	IF ncounter = nCount THEN 
		FOR i := 0 TO SIZEOF(refArray)-1 BY 1 DO 
			refArray[i] := FALSE;
		END_FOR
		F_checkMoveFinish := TRUE;
	ELSE
		F_checkMoveFinish := FALSE;
	END_IF
ELSE
	FOR i := 0 TO SIZEOF(refArray)-1 BY 1 DO 
			refArray[i] := FALSE;
		END_FOR
		F_checkMoveFinish := TRUE;
END_IF

END_FUNCTION

// ---- POUs/PROGRAMS/eflex.TcPOU
PROGRAM eflex
VAR
fbMqttClient	: FB_IotMqttClient;


bSetParameter 	: BOOL := TRUE;
bConnect 		: BOOL := TRUE;

(* published message *)
bPublish 		: BOOL;
sTopicPub 		: STRING(255) := 'flipper2.1toNodeRed'; //Publish topic. Must match syntax of nodeRed "mqtt out - topic"
sPayloadPub 	: STRING (255):= 'This is a test';
x				: UDINT;

(* recieved message *)
bSubscribed 	: BOOL;
sTopicSub 		: STRING(255) := 'toFlipper2.1PLC'; //Suscribe topic. Must match syntax of nodeRed "mqtt in - topic"
sTopicRcv 		: STRING(255);
sPayloadRcv 	: STRING(255);

fbMessageQueue	: FB_IotMqttMessageQueue;
fbMessage		: FB_IotMqttMessage;
fbJsonDataType 	: FB_JsonReadWriteDataType;
eflexMsgIn 		: ST_eflexMsgIn; //Custom Data Structure that must match variable types of eflex variables being sent through nodeRed. 
sBuffer 		: STRING(255);
END_VAR

IF bSetParameter THEN
	bSetParameter 				:= FALSE;
	fbMqttClient.sHostName 		:= '10.0.0.41';
	fbMqttClient.nHostPort 		:= 1883;
	fbMqttClient.sUserName 		:= 'eflex';
	fbMqttClient.sUserPassword 	:= 'dean-wormwood-sway-lope';
	fbMqttClient.ipMessageQueue := fbMessageQueue;
END_IF

fbMqttClient.Execute(bConnect);


IF fbMqttClient.bConnected THEN
	IF NOT bSubscribed THEN
		bSubscribed 	:= fbMqttClient.Subscribe(sTopic := sTopicSub, eQoS:= TcIOTMqttQos.AtMostOnceDelivery);
	END_IF
	IF bPublish THEN
		fbMqttClient.Publish(
		sTopic			:= sTopicPub, 
		pPayload		:= ADR(sBuffer), 
		nPayloadSize	:= LEN2(ADR(sBuffer)), 
		eQoS			:= TcIOTMqttQos.AtMostOnceDelivery, 
		bRetain			:= FALSE, 
		bQueue			:= FALSE);
		bPublish 		:= FALSE;	
		x := MEMSET(destAddr := ADR(sPayloadRcv),fillByte := 0,n := SIZEOF(sPayloadRcv));			
	END_IF
END_IF

IF fbMessageQueue.nQueuedMessages > 0 THEN 
	IF fbMessageQueue.Dequeue(fbMessage := fbMessage) THEN
		fbMessage.GetTopic(pTopic := ADR(sTopicRcv), nTopicSize := SIZEOF(sTopicRcv));
		fbMessage.GetPayload(pPayload:=ADR(sPayloadRcv), nPayloadSize:=SIZEOF(sPayloadRcv), bSetNullTermination:=FALSE);
		fbJsonDataType.SetSymbolFromJson(sPayloadRcv,'ST_eflexMsgIn',SIZEOF(eflexMsgIn), ADR(eflexMsgIn));
		GVL_eflex.bEflexPresent := TRUE;
		GVL_eflex.fFlipHeight := eflexMsgIn.flipHeight;
		GVL_eflex.fStudHeight := eflexMsgIn.studHeight;
		GVL_eflex.sSpaModel := eflexMsgIn.spaModel;
		GVL_eflex.fBaseInHeight := eflexMsgIn.baseInHeight;
		GVL_eflex.fSpaOutHeight := eflexMsgIn.spaOutHeight;
		sBuffer := fbJsonDataType.GetJsonStringFromSymbol('ST_eflexMsgIn',SIZEOF(eflexMsgIn), ADR(eflexMsgIn));
		bPublish := TRUE;
	END_IF
END_IF

IF GVL_eflex.bEflexPresent THEN
	IF GVL_eflex.fFlipHeight < 1 OR GVL_eflex.fStudHeight < 1 OR GVL_eflex.sSpaModel = '' THEN
		GVL_eflex.sSpaModel := 'ERROR';
	END_IF
END_IF

END_PROGRAM

// ---- POUs/PROGRAMS/tempEflex.TcPOU
PROGRAM tempEflex
VAR
	//HMI
	nEflexState : INT;
END_VAR



CASE nEflexState OF 
	0://Steady State
	1://A5L
		GVL_eflex.fBaseInHeight := 30;
		GVL_eflex.fSpaOutHeight := 35;
		GVL_eflex.fFlipHeight := 19;
		GVL_eflex.fStudHeight := 7;
		GVL_eflex.sSpaModel := 'A5L';
		GVL_eflex.bEflexPresent := TRUE;
		nEflexState := 0;
	2://A6
		GVL_eflex.fBaseInHeight := 30;
		GVL_eflex.fSpaOutHeight := 35;
		GVL_eflex.fFlipHeight := 22;
		GVL_eflex.fStudHeight := 12;
		GVL_eflex.sSpaModel := 'A6';
		GVL_eflex.bEflexPresent := TRUE;
		nEflexState := 0;
	3://A7
		GVL_eflex.fBaseInHeight := 30;
		GVL_eflex.fSpaOutHeight := 35;
		GVL_eflex.fFlipHeight := 23;
		GVL_eflex.fStudHeight := 12;
		GVL_eflex.sSpaModel := 'A7';
		GVL_eflex.bEflexPresent := TRUE;
		nEflexState := 0;
	4://A8
		GVL_eflex.fBaseInHeight := 27.5;
		GVL_eflex.fSpaOutHeight := 35;
		GVL_eflex.fFlipHeight := 24;
		GVL_eflex.fStudHeight := 15.5;
		GVL_eflex.sSpaModel := 'A8';
		GVL_eflex.bEflexPresent := TRUE;
		nEflexState := 0;
	5://A9L
		GVL_eflex.fBaseInHeight := 20.5;
		GVL_eflex.fSpaOutHeight := 35;
		GVL_eflex.fFlipHeight := 24;
		GVL_eflex.fStudHeight := 14.5;
		GVL_eflex.sSpaModel := 'A9L';
		GVL_eflex.bEflexPresent := TRUE;
		nEflexState := 0;
END_CASE

END_PROGRAM

// ---- POUs/PROGRAMS/motorsInit.TcPOU
PROGRAM motorsInit
VAR
	nInitCount	: INT;
	bChecked 	: BOOL := FALSE;
	nWaitCount 	: INT;
	aMoveFinish	: ARRAY[0..10] OF BOOL; // Can track the completion of up to 10 simultaneous moves
	fbMotorTimeOut : TON;
	fbWaitInit : TON;
	bMotorsInit : BOOL;
END_VAR

	updateMotors();
bMotorsInit := FALSE;
fbWaitInit(IN:= TRUE, PT:=T#3S);
fbMotorTimeOut(PT:=T#1M);

IF fbWaitInit.Q THEN
		GVL_machine.bMotorInitFailedDisp := FALSE;
		
		IF NOT aMoveFinish[1] THEN
			aMoveFinish[1] := GVL_devices.fbColumn1Motor.init(
								bMotorInvertedIn:= TRUE, 
								bMotorDisablesIn:= FALSE, 
								fMoveAcclIn:= 200, 
								fMoveDclIn:= 200, 
								fMoveVelocityIn:= 10, 
								torqueVelocityIn:= 10, 
								torqueAccelerationIn:= 50, 
								torqueDecelerationIn:= 50, 
								homeVelocityIn:= 7, 
								homeSetPositionIn:= 0, 
								homeTorqueLimitIn:= 8,
								jogTorqueIn := 100,
								bHasHomeSensorIn := FALSE);
		END_IF
		IF NOT aMoveFinish[2] THEN
			aMoveFinish[2] := GVL_devices.fbColumn2Motor.init(
								bMotorInvertedIn:= TRUE, 
								bMotorDisablesIn:= FALSE, 
								fMoveAcclIn:= 200, 
								fMoveDclIn:= 200, 
								fMoveVelocityIn:= 10, 
								torqueVelocityIn:= 10, 
								torqueAccelerationIn:= 50, 
								torqueDecelerationIn:= 50, 
								homeVelocityIn:= 7, 
								homeSetPositionIn:= 0, 
								homeTorqueLimitIn:= 8,
								jogTorqueIn := 100,
								bHasHomeSensorIn := TRUE);
		END_IF
		IF NOT aMoveFinish[3] THEN
			aMoveFinish[3] := GVL_devices.fbColumn3Motor.init(
								bMotorInvertedIn:= TRUE, 
								bMotorDisablesIn:= FALSE, 
								fMoveAcclIn:= 200, 
								fMoveDclIn:= 200, 
								fMoveVelocityIn:= 10, 
								torqueVelocityIn:= 10, 
								torqueAccelerationIn:= 50, 
								torqueDecelerationIn:= 50, 
								homeVelocityIn:= 7, 
								homeSetPositionIn:= 0, 
								homeTorqueLimitIn:= 8,
								jogTorqueIn := 100,
								bHasHomeSensorIn := FALSE);
		END_IF
		IF NOT aMoveFinish[4] THEN
			aMoveFinish[4] := GVL_devices.fbLftClampMotor.init(
								bMotorInvertedIn:= TRUE, 
								bMotorDisablesIn:= TRUE, 
								fMoveAcclIn:= 100, 
								fMoveDclIn:= 100, 
								fMoveVelocityIn:= 20, 
								torqueVelocityIn:= 7, 
								torqueAccelerationIn:= 100, 
								torqueDecelerationIn:= 100, 
								homeVelocityIn:= 10, 
								homeSetPositionIn:= 0, 
								homeTorqueLimitIn:= 20,
								jogTorqueIn := GVL_persistent.fTempLftClampTorque,
								bHasHomeSensorIn := FALSE);
		END_IF
		IF NOT aMoveFinish[5] THEN
			aMoveFinish[5] := GVL_devices.fbRhtClampMotor.init(
								bMotorInvertedIn:= FALSE, 
								bMotorDisablesIn:= TRUE, 
								fMoveAcclIn:= 100, 
								fMoveDclIn:= 100, 
								fMoveVelocityIn:= 20, 
								torqueVelocityIn:= 7, 
								torqueAccelerationIn:= 100, 
								torqueDecelerationIn:= 100, 
								homeVelocityIn:= 10, 
								homeSetPositionIn:= 0, 
								homeTorqueLimitIn:= 40,
								jogTorqueIn := GVL_persistent.fClampOnTorque,
								bHasHomeSensorIn := FALSE);
		END_IF
		IF NOT aMoveFinish[6] THEN
			aMoveFinish[6] := GVL_devices.fbLftRotationMotor.init(
								bMotorInvertedIn:= TRUE, 
								bMotorDisablesIn:= TRUE, 
								fMoveAcclIn:= 50, 
								fMoveDclIn:= 50, 
								fMoveVelocityIn:= 8, 
								torqueVelocityIn:= 7, 
								torqueAccelerationIn:= 50, 
								torqueDecelerationIn:= 50, 
								homeVelocityIn:= 3, 
								homeSetPositionIn:= GVL_persistent.fLftRotationHomePos, 
								homeTorqueLimitIn:= 20,
								jogTorqueIn := 100,
								bHasHomeSensorIn := FALSE);
		END_IF
		IF NOT aMoveFinish[7] THEN
			aMoveFinish[7] := GVL_devices.fbRhtRotationMotor.init(
								bMotorInvertedIn:= FALSE, 
								bMotorDisablesIn:= TRUE, 
								fMoveAcclIn:= 50, 
								fMoveDclIn:= 50, 
								fMoveVelocityIn:= 8, 
								torqueVelocityIn:= 7, 
								torqueAccelerationIn:= 50, 
								torqueDecelerationIn:= 50, 
								homeVelocityIn:= 3, 
								homeSetPositionIn:= GVL_persistent.fRhtRotationHomePos,
								homeTorqueLimitIn:= 20,
								jogTorqueIn := 100,
								bHasHomeSensorIn := FALSE);
		END_IF
		IF NOT aMoveFinish[8] THEN
			aMoveFinish[8] := GVL_devices.fbLftWidthMotor.init(
								bMotorInvertedIn:= FALSE, 
								bMotorDisablesIn:= TRUE, 
								fMoveAcclIn:= 50, 
								fMoveDclIn:= 50, 
								fMoveVelocityIn:= 20, 
								torqueVelocityIn:= 20, 
								torqueAccelerationIn:= 50, 
								torqueDecelerationIn:= 50, 
								homeVelocityIn:= 10, 
								homeSetPositionIn:= 0, 
								homeTorqueLimitIn:= 15,
								jogTorqueIn := 30,
								bHasHomeSensorIn := TRUE);
		END_IF
		IF NOT aMoveFinish[9] THEN
			aMoveFinish[9] := GVL_devices.fbRhtWidthMotor.init(
								bMotorInvertedIn:= FALSE, 
								bMotorDisablesIn:= TRUE, 
								fMoveAcclIn:= 50, 
								fMoveDclIn:= 50, 
								fMoveVelocityIn:= 20, 
								torqueVelocityIn:= 20, 
								torqueAccelerationIn:= 50, 
								torqueDecelerationIn:= 50, 
								homeVelocityIn:= 10, 
								homeSetPositionIn:= 0, 
								homeTorqueLimitIn:= 15,
								jogTorqueIn := 30,
								bHasHomeSensorIn := TRUE);
		END_IF
		IF NOT aMoveFinish[0] THEN
			aMoveFinish[0] := GVL_devices.fbColumn0Motor.init(
								bMotorInvertedIn:= TRUE, 
								bMotorDisablesIn:= FALSE, 
								fMoveAcclIn:= 200, 
								fMoveDclIn:= 200, 
								fMoveVelocityIn:= 10, 
								torqueVelocityIn:= 10, 
								torqueAccelerationIn:= 50, 
								torqueDecelerationIn:= 50, 
								homeVelocityIn:= 7, 
								homeSetPositionIn:= 0, 
								homeTorqueLimitIn:= 8,
								jogTorqueIn := 100,
								bHasHomeSensorIn := TRUE);
		END_IF
		
		IF F_checkMoveFinish(aMoveFinish,10,FALSE) THEN
			GVL_machine.sMotorInitState := 'PASSED';
			fbWaitInit(IN := FALSE);
			fbMotorTimeOut(IN := FALSE);
			GVL_machine.bMotorInitFailedDisp := FALSE;
			GVL_machine.bMotorsInitialized := TRUE;
			bMotorsInit := TRUE;
		ELSE // Start Timeout Timer
			fbMotorTimeout.IN := TRUE;
			IF fbMotorTimeout.Q THEN
				fbWaitInit(IN := FALSE);
				fbMotorTimeOut(IN := FALSE);
				GVL_machine.sMotorInitState := 'FAILED';
				GVL_machine.bMotorInitFailedDisp := TRUE;
				F_checkMoveFinish(aMoveFinish,10,TRUE);
				GVL_machine.bMotorsInitialized := TRUE;
			END_IF
		END_IF
	IF LEN(GVL_machine.sMotorInitState) <> 0 THEN
		GVL_devices.fbLftClampMotor.brakeOn();
		GVL_devices.fbRhtClampMotor.brakeOn();
	END_IF
END_IF

END_PROGRAM

// ---- POUs/PROGRAMS/updateMotors.TcPOU
PROGRAM updateMotors
VAR
END_VAR

GVL_devices.fbLftWidthMotor();
GVL_devices.fbRhtWidthMotor();

GVL_devices.fbLftClampMotor();
GVL_devices.fbRhtClampMotor();

GVL_devices.fbLftRotationMotor();	
GVL_devices.fbRhtRotationMotor();	

GVL_devices.fbColumn0Motor();	
GVL_devices.fbColumn1Motor();	
GVL_devices.fbColumn2Motor();	
GVL_devices.fbColumn3Motor();

END_PROGRAM

// ---- POUs/PROGRAMS/manual.TcPOU
PROGRAM manual
VAR
	aMoveFinishRotation			: ARRAY[0..10] OF BOOL; // Can track the completion of up to 10 simultaneous moves
	aMoveFinishColumn			: ARRAY[0..10] OF BOOL; // Can track the completion of up to 10 simultaneous moves
	aMoveFinishClamping			: ARRAY[0..10] OF BOOL; // Can track the completion of up to 10 simultaneous moves
	aMoveFinishWidth			: ARRAY[0..10] OF BOOL; // Can track the completion of up to 10 simultaneous moves
	
	eRotationState 	: E_manualState;
	eColumnState 	: E_manualState;
	eClampingState	: E_manualState;
	eWidthState		: E_manualState;
	eTableState		: E_manualState;
	
	fbCoupledRotation : TON;
	fbCoupledColumn : TON;
	fbCoupledClamping : TON;
	fbCoupledWidth : TON;
	tUncoupledTimeout : TIME := T#500MS;
	
	bRotationStopped 	: BOOL;
	bColumnStopped 		: BOOL;
	bClampingStopped 	: BOOL;
	bWidthStopped 		: BOOL;
	bTableStopped		: BOOL;
	
	//HMI 
	bHideRotationBtns 	: BOOL;
	bHideColumnBtns 	: BOOL;
	bHideClampingBtns	: BOOL;
	bHideWidthBtns		: BOOL;
	bHideTableBtns		: BOOL;
	
	bRotationMoveStatus : BOOL; // True- error is present
	bColumnMoveStatus 	: BOOL;
	bClampingMoveStatus : BOOL;
	bWidthMoveStatus 	: BOOL;
	bTableMoveStatus 	: BOOL;
	writeParameter		: MC_AxisParameter;
END_VAR

// Both manualScreen and manualBypassedScreen use this program for their functionality. Only difference is buttons are not hidden on manualBypassedScreen. 
///////////////////////// PAGE CHANGE TO MANUAL //////////////////////////////
IF GVL_machine.bPageChange THEN 
	eRotationState 	:= STEADYSTATE;
	eColumnState 	:= STEADYSTATE;
	eClampingState 	:= STEADYSTATE;
	eWidthState 	:= STEADYSTATE;
	eTableState		:= STEADYSTATE;
	GVL_machine.bPageChange	:= FALSE;
END_IF

fbCoupledRotation(PT := tUncoupledTimeout);
fbCoupledColumn(PT := tUncoupledTimeout); 
fbCoupledClamping (PT := tUncoupledTimeout);
fbCoupledWidth (PT := tUncoupledTimeout);


IF GVL_machine.bMuteSafety OR GVL_machine.bSafetyBypass THEN
	//pass -default is yellow
ELSIF bRotationStopped AND bColumnStopped AND bClampingStopped AND bWidthStopped AND bTableStopped THEN
	GVL_devices.fbLtCurtains.mute();
	IF GVL_devices.fbLtCurtains.curtainsMuted THEN
		GVL_devices.fbLtBars.greenOn();
	END_IF
ELSIF NOT bRotationStopped OR NOT bColumnStopped OR NOT bClampingStopped OR NOT bWidthStopped OR NOT bTableStopped THEN
	GVL_devices.fbLtBars.redOn();
END_IF




IF NOT GVL_machine.bSafetyOk AND NOT GVL_machine.bSafetyBypass THEN 
	GVL_devices.fbLtBars.redOn();
	GVL_devices.fbColumn0Motor.estop();
	GVL_devices.fbColumn1Motor.estop();
	GVL_devices.fbColumn2Motor.estop();
	GVL_devices.fbColumn3Motor.estop();
	GVL_devices.fbLftClampMotor.estop();
	GVL_devices.fbRhtClampMotor.estop();
	GVL_devices.fbLftRotationMotor.estop();
	GVL_devices.fbRhtRotationMotor.estop();
	GVL_devices.fbLftWidthMotor.estop();
	GVL_devices.fbRhtWidthMotor.estop();
	GVL_devices.fbTable.estop();
	eRotationState 	:= STEADYSTATE;
	eColumnState 	:= STEADYSTATE;
	eClampingState 	:= STEADYSTATE;
	eWidthState 	:= STEADYSTATE;
	
ELSE // No Estop or Light Curtain 
	(*				Rotation Motion 			*)
		bRotationStopped := FALSE;
		bHideRotationBtns := TRUE;
		CASE eRotationState OF 
			STEADYSTATE:
				bHideRotationBtns := FALSE;
				bRotationStopped := TRUE;
				fbCoupledRotation.IN := FALSE;
				bRotationMoveStatus := FALSE;
				F_checkMoveFinish(aMoveFinishRotation,1,TRUE);
				
			MOVEAWAYDIRECTION:
				bHideRotationBtns := FALSE;
				CASE GVL_devices.fbLftRotationMotor.moveToJog(0) OF 
					1: // Good
					13://Error
						bRotationMoveStatus := TRUE; 
						GVL_machine.motorErrorList := LFTROTATION;
						GVL_machine.bErrorPresent := TRUE;
				END_CASE
				CASE GVL_devices.fbRhtRotationMotor.moveToJog(1) OF
					1: // Good
					13://Error
						bRotationMoveStatus := TRUE;
						GVL_machine.motorErrorList := RHTROTATION;
						GVL_machine.bErrorPresent := TRUE; 
				END_CASE
				CASE F_checkCoupledMovement(GVL_devices.fbLftRotationMotor.fbMotor,GVL_devices.fbRhtRotationMotor.fbMotor) OF 
						0: fbCoupledRotation.IN := FALSE;
						1,2: fbCoupledRotation.IN := TRUE;
						3: fbCoupledRotation.IN := FALSE;
				END_CASE
				
			MOVEHOMEDIRECTION:
				bHideRotationBtns := FALSE;
				CASE GVL_devices.fbLftRotationMotor.moveToJog(1) OF
					1: // Good
					13://Error
						bRotationMoveStatus := TRUE;
						GVL_machine.motorErrorList := LFTROTATION;
						GVL_machine.bErrorPresent := TRUE; 
				END_CASE
				CASE GVL_devices.fbRhtRotationMotor.moveToJog(0) OF
					1: // Good
					13://Error
						bRotationMoveStatus := TRUE; 
						GVL_machine.motorErrorList := RHTROTATION;
						GVL_machine.bErrorPresent := TRUE; 
				END_CASE
				CASE F_checkCoupledMovement(GVL_devices.fbLftRotationMotor.fbMotor,GVL_devices.fbRhtRotationMotor.fbMotor) OF 
						0: fbCoupledRotation.IN := FALSE;
						1,2: fbCoupledRotation.IN := TRUE;
						3: fbCoupledRotation.IN := FALSE;
				END_CASE
				
			RESET:
				IF NOT aMoveFinishRotation[0] THEN
					CASE GVL_devices.fbLftRotationMotor.reset() OF
						1:// Done
							aMoveFinishRotation[0] := TRUE;
						13:// Error
							bRotationMoveStatus := TRUE;
							GVL_machine.motorErrorList := LFTROTATION;
							GVL_machine.bErrorPresent := TRUE;
					END_CASE
				END_IF
				IF NOT aMoveFinishRotation[1] THEN
					CASE GVL_devices.fbRhtRotationMotor.reset() OF
						1:// Done
							aMoveFinishRotation[1] := TRUE;
						13:// Error
							bRotationMoveStatus := TRUE;
							GVL_machine.motorErrorList := RHTROTATION;
							GVL_machine.bErrorPresent := TRUE; 
						
					END_CASE 
				END_IF
				IF F_checkMoveFinish(aMoveFinishRotation,2,FALSE) THEN
					bRotationMoveStatus := FALSE;
					eRotationState := STEADYSTATE;
				END_IF
				
			HOMING:
				IF GVL_devices.fbLftRotationMotor.fbMotor.Status.Homed AND GVL_devices.fbRhtRotationMotor.fbMotor.Status.Homed THEN
					CASE F_checkCoupledMovement(GVL_devices.fbLftRotationMotor.fbMotor,GVL_devices.fbRhtRotationMotor.fbMotor) OF 
						0: fbCoupledRotation.IN := FALSE;
						1,2: fbCoupledRotation.IN := TRUE;
						3: fbCoupledRotation.IN := FALSE;
					END_CASE
				END_IF
				IF NOT aMoveFinishRotation[0] THEN
					CASE GVL_devices.fbLftRotationMotor.homeToTorque() OF 
						1:// Done
							aMoveFinishRotation[0] := TRUE;
						13:// Error
							GVL_machine.motorErrorList := LFTROTATION;
							GVL_machine.bErrorPresent := TRUE;
					END_CASE
				END_IF
				IF NOT aMoveFinishRotation[1] THEN
					CASE GVL_devices.fbRhtRotationMotor.homeToTorque() OF 
						1:// Done
							aMoveFinishRotation[1] := TRUE;
						13:// Error
							GVL_machine.motorErrorList := RHTROTATION;
							GVL_machine.bErrorPresent := TRUE; 
					END_CASE
				END_IF
				IF F_checkMoveFinish(aMoveFinishRotation,2,FALSE) THEN
					eRotationState := STEADYSTATE;
				END_IF
		END_CASE
		
		//Initial Homing not done or Components not moving together
		IF NOT GVL_devices.fbLftRotationMotor.fbMotor.Status.Homed OR NOT GVL_devices.fbRhtRotationMotor.fbMotor.Status.Homed OR fbCoupledRotation.Q OR bRotationMoveStatus THEN	
			GVL_devices.fbLftRotationMotor.estop();
			GVL_devices.fbRhtRotationMotor.estop();
			bHideRotationBtns := TRUE;
		END_IF
		
	(*				Column Motion 				*)
		bColumnStopped := FALSE;
		bHideColumnBtns := TRUE;
		CASE eColumnState OF 
			STEADYSTATE:
				bHideColumnBtns := FALSE;
				bColumnStopped := TRUE;
				fbCoupledColumn.IN := FALSE;
				bColumnMoveStatus := FALSE;
				F_checkMoveFinish(aMoveFinishColumn,1,TRUE);
				
			MOVEAWAYDIRECTION:
				bHideColumnBtns := FALSE;
				IF GVL_devices.fbColumn1Motor.fbMotor.Status.Coupled AND GVL_devices.fbColumn2Motor.fbMotor.Status.Coupled AND GVL_devices.fbColumn3Motor.fbMotor.Status.Coupled THEN
					GVL_devices.fbColumn0Motor.motorIdle := FALSE;
					GVL_devices.fbColumn1Motor.motorIdle := FALSE;
					GVL_devices.fbColumn2Motor.motorIdle := FALSE;
					GVL_devices.fbColumn3Motor.motorIdle := FALSE;
					CASE GVL_devices.fbColumn0Motor.moveToJog(0) OF
						1:// Good
						13:// Error
							bColumnMoveStatus := TRUE;
							GVL_machine.motorErrorList := COLUMN0;
							GVL_machine.bErrorPresent := TRUE; 
					END_CASE
				ELSE // Couple Motors
					GVL_devices.fbColumn1Motor.coupleToAxis(GVL_devices.fbColumn0Motor.fbMotor);
					GVL_devices.fbColumn2Motor.coupleToAxis(GVL_devices.fbColumn0Motor.fbMotor);
					GVL_devices.fbColumn3Motor.coupleToAxis(GVL_devices.fbColumn0Motor.fbMotor);
				END_IF
				
			MOVEHOMEDIRECTION:
				bHideColumnBtns := FALSE;
				
				
				IF GVL_devices.fbColumn1Motor.fbMotor.Status.Coupled AND GVL_devices.fbColumn2Motor.fbMotor.Status.Coupled AND GVL_devices.fbColumn3Motor.fbMotor.Status.Coupled THEN
					GVL_devices.fbColumn0Motor.motorIdle := FALSE;
					GVL_devices.fbColumn1Motor.motorIdle := FALSE;
					GVL_devices.fbColumn2Motor.motorIdle := FALSE;
					GVL_devices.fbColumn3Motor.motorIdle := FALSE;
					CASE GVL_devices.fbColumn0Motor.moveToJog(1) OF 
						1:// Good
						13:// Error
							bColumnMoveStatus := TRUE;
							GVL_machine.motorErrorList := COLUMN0;
							GVL_machine.bErrorPresent := TRUE; 
					END_CASE
				ELSE // Couple Motors
					GVL_devices.fbColumn1Motor.coupleToAxis(GVL_devices.fbColumn0Motor.fbMotor);
					GVL_devices.fbColumn2Motor.coupleToAxis(GVL_devices.fbColumn0Motor.fbMotor);
					GVL_devices.fbColumn3Motor.coupleToAxis(GVL_devices.fbColumn0Motor.fbMotor);
				END_IF
			RESET:
				IF NOT aMoveFinishColumn[0] THEN
					CASE GVL_devices.fbColumn0Motor.reset() OF 
						1:// Done
							aMoveFinishColumn[0] := TRUE;
						13:// Error
							bColumnMoveStatus := TRUE;
							GVL_machine.motorErrorList := COLUMN0;
							GVL_machine.bErrorPresent := TRUE; 
					END_CASE
				END_IF
				IF NOT aMoveFinishColumn[1] THEN
					CASE GVL_devices.fbColumn1Motor.reset() OF 
						1:// Done
							aMoveFinishColumn[1] := TRUE;
						13:// Error
							bColumnMoveStatus := TRUE;
							GVL_machine.motorErrorList := COLUMN1;
							GVL_machine.bErrorPresent := TRUE; 
					END_CASE
				END_IF
				IF NOT aMoveFinishColumn[2] THEN
					CASE GVL_devices.fbColumn2Motor.reset() OF 
						1:// Done
							aMoveFinishColumn[2] := TRUE;
						13:// Error
							bColumnMoveStatus := TRUE;
							GVL_machine.motorErrorList := COLUMN2;
							GVL_machine.bErrorPresent := TRUE; 
					END_CASE
				END_IF
				IF NOT aMoveFinishColumn[3] THEN
					CASE GVL_devices.fbColumn3Motor.reset() OF 
						1:// Done
							aMoveFinishColumn[3] := TRUE;
						13:// Error
							bColumnMoveStatus := TRUE;
							GVL_machine.motorErrorList := COLUMN3;
							GVL_machine.bErrorPresent := TRUE; 
					END_CASE
				END_IF
				
				IF F_checkMoveFinish(aMoveFinishColumn,4,FALSE) THEN
					eColumnState := STEADYSTATE;
				END_IF
				
			HOMING:
				(*IF GVL_devices.fbColumn0Motor.fbMotor.Status.Homed AND GVL_devices.fbColumn2Motor.fbMotor.Status.Homed THEN
					writeParameter := AxisMaxSoftPosLimit;
					IF NOT aMoveFinishColumn[0] THEN
						CASE GVL_devices.fbColumn2Motor.writeRealParameter(writeParameter,1) OF 
							1: //Done
								aMoveFinishColumn[0] := TRUE;
							13:// Error
								bColumnMoveStatus := TRUE;
								GVL_machine.motorErrorList := COLUMN2;
								GVL_machine.bErrorPresent := TRUE; 
						END_CASE
					END_IF
					IF aMoveFinishColumn[0] AND NOT aMoveFinishColumn[1] THEN
						IF GVL_devices.fbColumn1Motor.fbMotor.Status.Coupled AND GVL_devices.fbColumn2Motor.fbMotor.Status.Coupled AND GVL_devices.fbColumn3Motor.fbMotor.Status.Coupled THEN
							GVL_devices.fbColumn0Motor.motorIdle := FALSE;
							GVL_devices.fbColumn1Motor.motorIdle := FALSE;
							GVL_devices.fbColumn2Motor.motorIdle := FALSE;
							GVL_devices.fbColumn3Motor.motorIdle := FALSE;
							CASE GVL_devices.fbColumn0Motor.homeToSensor(0) OF 
								1: // Done
									aMoveFinishColumn[1] := TRUE;
								13:// Error
									bColumnMoveStatus := TRUE;
									GVL_machine.motorErrorList := COLUMN0;
									GVL_machine.bErrorPresent := TRUE; 
							END_CASE
						ELSE // Couple Motors to Column0
							GVL_devices.fbColumn1Motor.coupleToAxis(GVL_devices.fbColumn0Motor.fbMotor);
							GVL_devices.fbColumn2Motor.coupleToAxis(GVL_devices.fbColumn0Motor.fbMotor);
							GVL_devices.fbColumn3Motor.coupleToAxis(GVL_devices.fbColumn0Motor.fbMotor);
						END_IF
					END_IF
					IF aMoveFinishColumn[1] AND NOT aMoveFinishColumn[2] THEN
						CASE GVL_devices.fbColumn2Motor.writeRealParameter(writeParameter,0) OF 
							1:// Done
								aMoveFinishColumn[2] := TRUE;
							13://Error
								bColumnMoveStatus := TRUE;
								GVL_machine.motorErrorList := COLUMN2;
								GVL_machine.bErrorPresent := TRUE; 
						END_CASE
					END_IF
					IF F_checkMoveFinish(aMoveFinishColumn,3,FALSE) THEN
						eColumnState := STEADYSTATE;
					END_IF
				ELSE
					IF NOT aMoveFinishColumn[0] THEN
						IF GVL_devices.fbColumn1Motor.fbMotor.Status.Coupled THEN
							GVL_devices.fbColumn0Motor.motorIdle := FALSE;
							GVL_devices.fbColumn1Motor.motorIdle := FALSE;
							CASE GVL_devices.fbColumn0Motor.homeToSensor(0) OF 
								1:// Done
									aMoveFinishColumn[0] := TRUE;
								13:// Error
									bColumnMoveStatus := TRUE;
									GVL_machine.motorErrorList := COLUMN0;
									GVL_machine.bErrorPresent := TRUE; 
							END_CASE
						ELSE
							GVL_devices.fbColumn1Motor.coupleToAxis(GVL_devices.fbColumn0Motor.fbMotor);
						END_IF
					END_IF
					
					IF NOT aMoveFinishColumn[1] THEN
						IF GVL_devices.fbColumn3Motor.fbMotor.Status.Coupled THEN
							GVL_devices.fbColumn2Motor.motorIdle := FALSE;
							GVL_devices.fbColumn3Motor.motorIdle := FALSE;
							CASE GVL_devices.fbColumn2Motor.homeToSensor(0) OF 
								1:// Done
									aMoveFinishColumn[1] := TRUE;
								13:// Error
									bColumnMoveStatus := TRUE;
									GVL_machine.motorErrorList := COLUMN2;
									GVL_machine.bErrorPresent := TRUE; 
							END_CASE
						ELSE
							GVL_devices.fbColumn3Motor.coupleToAxis(GVL_devices.fbColumn2Motor.fbMotor);
						END_IF
					END_IF
					
					IF F_checkMoveFinish(aMoveFinishColumn,2,FALSE) THEN
						eColumnState := STEADYSTATE;
					END_IF
					
				END_IF*)
				IF NOT aMoveFinishColumn[0] THEN
					IF GVL_devices.fbColumn1Motor.fbMotor.Status.Coupled THEN
						GVL_devices.fbColumn0Motor.motorIdle := FALSE;
						GVL_devices.fbColumn1Motor.motorIdle := FALSE;
						CASE GVL_devices.fbColumn0Motor.homeToSensor(0) OF 
							1:// Done
								aMoveFinishColumn[0] := TRUE;
							13:// Error
								GVL_machine.motorErrorList := COLUMN0;
								GVL_machine.bErrorPresent := TRUE;
						END_CASE
					ELSE
						CASE GVL_devices.fbColumn1Motor.coupleToAxis(GVL_devices.fbColumn0Motor.fbMotor) OF 
							1:// Done
							13: GVL_devices.fbColumn1Motor.reset();
								GVL_machine.motorErrorList := COLUMN1;
								GVL_machine.bErrorPresent := TRUE;
						END_CASE
					END_IF
				END_IF
				
				IF NOT aMoveFinishColumn[1] THEN
					IF GVL_devices.fbColumn3Motor.fbMotor.Status.Coupled THEN
						GVL_devices.fbColumn2Motor.motorIdle := FALSE;
						GVL_devices.fbColumn3Motor.motorIdle := FALSE;
						CASE GVL_devices.fbColumn2Motor.homeToSensor(0) OF 
							1:// Done
								aMoveFinishColumn[1] := TRUE;
							13://Error
								GVL_machine.motorErrorList := COLUMN2;
								GVL_machine.bErrorPresent := TRUE;
						END_CASE
					ELSE
						CASE GVL_devices.fbColumn3Motor.coupleToAxis(GVL_devices.fbColumn2Motor.fbMotor) OF 
							1://Done 
							13: GVL_devices.fbColumn3Motor.reset();
								GVL_machine.motorErrorList := COLUMN3;
								GVL_machine.bErrorPresent := TRUE;
						END_CASE
					END_IF
				END_IF
				
				IF F_checkMoveFinish(aMoveFinishColumn,2,FALSE) THEN
					eColumnState := STEADYSTATE;
				END_IF
		END_CASE
		
		//Initial Homing not done or Components not moving together
		IF NOT GVL_devices.fbColumn0Motor.fbMotor.Status.Homed OR NOT GVL_devices.fbColumn2Motor.fbMotor.Status.Homed OR fbCoupledColumn.Q THEN	
			bHideColumnBtns := TRUE;
		END_IF
		
	(* 				Clamping Motion				*)
		bClampingStopped := FALSE;
		bHideClampingBtns := TRUE;
		CASE eClampingState OF 
			STEADYSTATE:
				bHideClampingBtns := FALSE;
			 	bClampingStopped := TRUE;
				bClampingMoveStatus := FALSE;
				F_checkMoveFinish(aMoveFinishClamping,1,TRUE);
				
			MOVEAWAYDIRECTION:
				bHideClampingBtns := FALSE;
				(*CASE GVL_devices.fbLftClampMotor.moveToJog(0) OF 
					1:// Good
					13:// Error
						bClampingMoveStatus := TRUE;
						GVL_machine.motorErrorList := LFTCLAMP;
						GVL_machine.bErrorPresent := TRUE; 
				END_CASE*)
				GVL_devices.fbLftClampMotor.tempCylinderOpen();
				
				CASE GVL_devices.fbRhtClampMotor.moveToJog(1) OF
					1:// Good
					13:// Error
						bClampingMoveStatus := TRUE;
						GVL_machine.motorErrorList := RHTCLAMP;
						GVL_machine.bErrorPresent := TRUE; 
				END_CASE
				
			MOVEHOMEDIRECTION: 
				bHideClampingBtns := FALSE;
				(*CASE GVL_devices.fbLftClampMotor.moveToJog(1) OF 
					1://Good
					13:// Error
						bClampingMoveStatus := TRUE;
						GVL_machine.motorErrorList := LFTCLAMP;
						GVL_machine.bErrorPresent := TRUE; 
				END_CASE*)
				GVL_devices.fbLftClampMotor.tempCylinderClose();
				
				CASE GVL_devices.fbRhtClampMotor.moveToJog(0) OF
					1:// Good
					13:// Error
						bClampingMoveStatus := TRUE;
						GVL_machine.motorErrorList := RHTCLAMP;
						GVL_machine.bErrorPresent := TRUE; 
				END_CASE
			
			RESET:
				IF NOT aMoveFinishClamping[0] THEN
					CASE GVL_devices.fbLftClampMotor.reset() OF
						1:// Done
							aMoveFinishClamping[0] := TRUE;
						13:// Error
							bClampingMoveStatus := TRUE;
							GVL_machine.motorErrorList := LFTCLAMP;
							GVL_machine.bErrorPresent := TRUE; 
					END_CASE
				END_IF
				IF NOT aMoveFinishClamping[1] THEN
					CASE GVL_devices.fbRhtClampMotor.reset() OF 
						1:// Done
							aMoveFinishClamping[1] := TRUE;
						13:// Error
							bClampingMoveStatus := TRUE;
							GVL_machine.motorErrorList := RHTCLAMP;
							GVL_machine.bErrorPresent := TRUE; 
					END_CASE
				END_IF
				IF F_checkMoveFinish(aMoveFinishClamping,2,FALSE) THEN
					eClampingState := STEADYSTATE;
				END_IF
				
			HOMING:
				IF NOT aMoveFinishClamping[0] THEN
					(*CASE GVL_devices.fbLftClampMotor.homeToTorque() OF 
						1:// Done
							aMoveFinishClamping[0] := TRUE;
						13:// Error
							bClampingMoveStatus := TRUE;
							GVL_machine.motorErrorList := LFTCLAMP;
							GVL_machine.bErrorPresent := TRUE; 
					END_CASE*)
					IF GVL_devices.fbLftClampMotor.tempCylinderClose() THEN
						aMoveFinishClamping[0] := TRUE;
					END_IF
				END_IF
				IF NOT aMoveFinishClamping[1] THEN
					CASE GVL_devices.fbRhtClampMotor.homeToTorque() OF 
						1:// Done
							aMoveFinishClamping[1] := TRUE;
						13:// Error
							bClampingMoveStatus := TRUE;
							GVL_machine.motorErrorList := RHTCLAMP;
							GVL_machine.bErrorPresent := TRUE; 
					END_CASE
				END_IF
				IF F_checkMoveFinish(aMoveFinishClamping,2,FALSE) THEN
					eClampingState := STEADYSTATE;
				END_IF
		END_CASE
		//Initial Homing not done or Components not moving together
		(*IF NOT GVL_devices.fbLftClampMotor.fbMotor.Status.Homed OR NOT GVL_devices.fbRhtClampMotor.fbMotor.Status.Homed OR fbCoupledClamping.Q THEN	
			bHideClampingBtns := TRUE;
		END_IF*)
		IF NOT GVL_devices.fbRhtClampMotor.fbMotor.Status.Homed OR fbCoupledClamping.Q THEN	
			bHideClampingBtns := TRUE;
		END_IF
		
	(*				Width Motion 				*)
		bWidthStopped := FALSE;
		bHideWidthBtns := TRUE;
		CASE eWidthState OF 
			STEADYSTATE : 
				bHideWidthBtns := FALSE;
			 	bWidthStopped := TRUE;
				F_checkMoveFinish(aMoveFinishWidth,1,TRUE);
				
			MOVEAWAYDIRECTION:
				bHideWidthBtns := FALSE;
				//GVL_devices.fbLftWidthMotor.motorIdle:= FALSE;
				//GVL_devices.fbRhtWidthMotor.motorIdle:= FALSE;
				CASE GVL_devices.fbLftWidthMotor.moveToJog(1) OF 
					1: //Good
					13:// Error 
						bWidthMoveStatus := TRUE;
						GVL_machine.motorErrorList := LFTWIDTH;
						GVL_machine.bErrorPresent := TRUE; 
				END_CASE
				CASE GVL_devices.fbRhtWidthMotor.moveToJog(1) OF 
					1: //Good
					13:// Error 
						bWidthMoveStatus := TRUE;
						GVL_machine.motorErrorList := RHTWIDTH;
						GVL_machine.bErrorPresent := TRUE; 
				END_CASE
				
			MOVEHOMEDIRECTION:
				bHideWidthBtns := FALSE;
				//GVL_devices.fbLftWidthMotor.motorIdle:= FALSE;
				//GVL_devices.fbRhtWidthMotor.motorIdle:= FALSE;
				CASE GVL_devices.fbLftWidthMotor.moveToJog(0) OF
					1: //Good
					13:// Error 
						bWidthMoveStatus := TRUE;
						GVL_machine.motorErrorList := LFTWIDTH;
						GVL_machine.bErrorPresent := TRUE; 
				END_CASE
				CASE GVL_devices.fbRhtWidthMotor.moveToJog(0) OF
					1: //Good
					13:// Error 
						bWidthMoveStatus := TRUE;
						GVL_machine.motorErrorList := RHTWIDTH;
						GVL_machine.bErrorPresent := TRUE; 
				END_CASE
				
			RESET: 
				IF NOT aMoveFinishWidth[0] THEN
					CASE GVL_devices.fbLftWidthMotor.reset() OF 
						1:// Done
							aMoveFinishWidth[0] := TRUE;
						13:// Error
							bWidthMoveStatus := TRUE;
							GVL_machine.motorErrorList := LFTWIDTH;
							GVL_machine.bErrorPresent := TRUE; 
					END_CASE
				END_IF
				IF NOT aMoveFinishWidth[1] THEN
					CASE GVL_devices.fbRhtWidthMotor.reset() OF 
						1:// Done
							aMoveFinishWidth[1] := TRUE;
						13:// Error	
							bWidthMoveStatus := TRUE;
							GVL_machine.motorErrorList := RHTWIDTH;
							GVL_machine.bErrorPresent := TRUE; 
					END_CASE
				END_IF
				IF F_checkMoveFinish(aMoveFinishWidth,2,FALSE) THEN
					eWidthState := STEADYSTATE;
				END_IF
				
			HOMING:
				IF NOT aMoveFinishWidth[0] THEN
					CASE GVL_devices.fbLftWidthMotor.homeToSensorCustom() OF 
						1:// Done
							aMoveFinishWidth[0] := TRUE;
						13:// Error
							bWidthMoveStatus := TRUE;
							GVL_machine.motorErrorList := LFTWIDTH;
							GVL_machine.bErrorPresent := TRUE; 
					END_CASE
				END_IF
				IF NOT aMoveFinishWidth[1] THEN
					CASE GVL_devices.fbRhtWidthMotor.homeToSensorCustom() OF 
						1:// Done
							aMoveFinishWidth[1] := TRUE;
						13:// Error	
							bWidthMoveStatus := TRUE;
							GVL_machine.motorErrorList := RHTWIDTH;
							GVL_machine.bErrorPresent := TRUE; 
					END_CASE
				END_IF
				IF F_checkMoveFinish(aMoveFinishWidth,2,FALSE) THEN
					eWidthState := STEADYSTATE;
				END_IF
		END_CASE
		//Initial Homing not done or Components not moving together
		IF NOT GVL_devices.fbLftWidthMotor.fbMotor.Status.Homed OR NOT GVL_devices.fbRhtWidthMotor.fbMotor.Status.Homed OR fbCoupledWidth.Q THEN	
			bHideWidthBtns := TRUE;
		END_IF
		
	(*				Table Motion				*)
		bTableStopped := FALSE;
		bHideTableBtns := TRUE;
		CASE eTableState OF 
			STEADYSTATE:
				bHideTableBtns := FALSE;
			 	bTableStopped := TRUE;
				GVL_devices.fbTable.tempSteadyState();
			MOVEAWAYDIRECTION:
				bHideTableBtns := FALSE;
				GVL_devices.fbTable.tempMoveUp();
			MOVEHOMEDIRECTION:
				bHideTableBtns := FALSE; 
				GVL_devices.fbTable.tempMoveDown();
			HOMING: 
				IF GVL_devices.fbTable.moveTo(GVL_persistent.fTableConveyorHeight) THEN
					eTableState := STEADYSTATE;
				END_IF
		END_CASE
END_IF

END_PROGRAM

// ---- POUs/FUNCTIONS/F_checkCoupledMovement.TcPOU
FUNCTION F_checkCoupledMovement : INT //0- No movement, 1-axis1 is moving, 2-axis2 is moving, 3- axis1 and axis2 are moving. 
VAR_INPUT
	axis1 : AXIS_REF;
	axis2 : AXIS_REF; 
END_VAR
VAR
END_VAR

F_checkCoupledMovement := 0;

IF axis1.Status.Moving AND NOT axis2.Status.Moving THEN
	F_checkCoupledMovement := 1;
ELSIF axis1.Status.Moving AND NOT axis2.Status.Moving THEN
	F_checkCoupledMovement := 2;
ELSIF axis1.Status.Moving AND axis2.Status.Moving THEN
	F_checkCoupledMovement := 3;
END_IF

END_FUNCTION

// ---- POUs/PROGRAMS/errorHandling.TcPOU
PROGRAM errorHandling
VAR
	bResetBtn : BOOL;
	bExitBtn : BOOL;
	
	sBlock : STRING;
	nID : UDINT;
	sMsg : STRING;
	sLoc : STRING;
	
	nPrevId: UDINT;
	sPrevBlock : STRING;
END_VAR

//Create Page for each component and show it in a frame
CASE GVL_machine.motorErrorList OF 
	LFTROTATION : //pass
		sLoc := 'LEFT ROTATION';
		sBlock := GVL_devices.fbLftRotationMotor.stError.errorLoc;
		nID := GVL_devices.fbLftRotationMotor.stError.errorId;
		sMsg := GVL_devices.fbLftRotationMotor.stError.errorMsg;
		
		
	
	LFTCLAMP: //pass
		sLoc := 'LEFT CLAMP';
		sBlock := GVL_devices.fbLftClampMotor.stError.errorLoc;
		nID := GVL_devices.fbLftClampMotor.stError.errorId;
		sMsg := GVL_devices.fbLftClampMotor.stError.errorMsg;
		
		
	
	COLUMN0: //pass
		sLoc := 'COLUMN 0';
		sBlock := GVL_devices.fbColumn0Motor.stError.errorLoc;
		nID := GVL_devices.fbColumn0Motor.stError.errorId;
		sMsg := GVL_devices.fbColumn0Motor.stError.errorMsg;
		
		
	
	COLUMN1: //pass
		sLoc := 'COLUMN 1';
		sBlock := GVL_devices.fbColumn1Motor.stError.errorLoc;
		nID := GVL_devices.fbColumn1Motor.stError.errorId;
		sMsg := GVL_devices.fbColumn1Motor.stError.errorMsg;
		
	
		
	LFTWIDTH: //pass
		sLoc := 'LEFT WIDTH';
		sBlock := GVL_devices.fbLftWidthMotor.stError.errorLoc;
		nID := GVL_devices.fbLftWidthMotor.stError.errorId;
		sMsg := GVL_devices.fbLftWidthMotor.stError.errorMsg;
		

		
	RHTWIDTH: //pass
		sLoc := 'RIGHT WIDTH';
		sBlock := GVL_devices.fbRhtWidthMotor.stError.errorLoc;
		nID := GVL_devices.fbRhtWidthMotor.stError.errorId;
		sMsg := GVL_devices.fbRhtWidthMotor.stError.errorMsg;
		
		
		
	COLUMN2: //pass
		sLoc := 'COLUMN 2';
		sBlock := GVL_devices.fbColumn2Motor.stError.errorLoc;
		nID := GVL_devices.fbColumn2Motor.stError.errorId;
		sMsg := GVL_devices.fbColumn2Motor.stError.errorMsg;
		
	
		
	COLUMN3: //pass
		sLoc := 'COLUMN 3';
		sBlock := GVL_devices.fbColumn3Motor.stError.errorLoc;
		nID := GVL_devices.fbColumn3Motor.stError.errorId;
		sMsg := GVL_devices.fbColumn3Motor.stError.errorMsg;
		
		
	
	RHTCLAMP: //pass
		sLoc := 'RIGHT CLAMP';
		sBlock := GVL_devices.fbRhtClampMotor.stError.errorLoc;
		nID := GVL_devices.fbRhtClampMotor.stError.errorId;
		sMsg := GVL_devices.fbRhtClampMotor.stError.errorMsg;
		
	
		
	RHTROTATION: //pass
		sLoc := 'RIGHT ROTATION';
		sBlock := GVL_devices.fbRhtRotationMotor.stError.errorLoc;
		nID := GVL_devices.fbRhtRotationMotor.stError.errorId;
		sMsg := GVL_devices.fbRhtRotationMotor.stError.errorMsg;
		
	CUSTOM: //pass
		sLoc := GVL_machine.sLoc;
		sBlock := GVL_machine.sBlock;
		nID := GVL_machine.nID;
		sMsg := GVL_machine.sMsg;

END_CASE

IF sBlock = sPrevBlock AND nID = nPrevID THEN
	GVL_machine.bErrorPresent := FALSE;
ELSE
	F_recordErrorData(sLoc,sBlock,nId,sMsg);
	GVL_machine.bErrorPresent := FALSE;
	sPrevBlock := sBlock;
	nPrevId := nID;
END_IF

END_PROGRAM

// ---- POUs/FUNCTIONS/F_recordErrorData.TcPOU
FUNCTION F_recordErrorData : BOOL
VAR_INPUT
	sLoc 	: STRING;
	sBlock 	: STRING;
	nID 	: UDINT;
	sMsg 	: STRING;
END_VAR
VAR
	fbGetSystemTime  : GETSYSTEMTIME;
    fileTime         : T_FILETIME;
    sTime            : STRING;
	sStringCombine0 : STRING;
	sStringCombine1 : STRING;
	sStringCombine2 : STRING;
	sStringCombine3 : STRING;
	sStringCombine4 : STRING;
	sStringCombine5 : STRING;



END_VAR

fbGetSystemTime(timeLoDW=>fileTime.dwLowDateTime, timeHiDW=>fileTime.dwHighDateTime );

	//Set time of event 
	GVL_machine.aErrorData[1,GVL_machine.nErrorDataRow] := SYSTEMTIME_TO_STRING( FILETIME_TO_SYSTEMTIME( fileTime ) );
	//Set Motor Location
	GVL_machine.aErrorData[2,GVL_machine.nErrorDataRow] :=sLoc;
	//Set Function Block Location
	GVL_machine.aErrorData[3,GVL_machine.nErrorDataRow] := sBlock;
	//Set Error ID 
	GVL_machine.aErrorData[4,GVL_machine.nErrorDataRow] := UDINT_TO_STRING(nID);
	//Set Message Error 
	IF sMsg = '' THEN
		CASE nID OF 
			0,1: sStringCombine0 := CONCAT( '0: ' , LREAL_TO_STRING(GVL_devices.fbColumn0Motor.fbMotor.NcToPlc.ActPos));
				 sStringCombine1 := CONCAT( ', 1: ' , LREAL_TO_STRING(GVL_devices.fbColumn1Motor.fbMotor.NcToPlc.ActPos));
				 sStringCombine2 := CONCAT(', 2: ' , LREAL_TO_STRING(GVL_devices.fbColumn2Motor.fbMotor.NcToPlc.ActPos));
				 sStringCombine3 := CONCAT(', 3: ' , LREAL_TO_STRING(GVL_devices.fbColumn3Motor.fbMotor.NcToPlc.ActPos));
				 sStringCombine3 := CONCAT(sStringCombine0,sStringCombine1);
				 sStringCombine4 := CONCAT(sStringCombine2,sStringCombine3);
				 sMsg := CONCAT(sStringCombine3,sStringCombine4);
				 sStringCombine0 := '';
				 sStringCombine1 := '';
				 sStringCombine2 := '';
				 sStringCombine3 := '';
				 sStringCombine3 := '';
				 sStringCombine4 := '';
			16992: sMsg := 'The master axis start position does not permit synchronization';
			17056: sMsg := 'Group/axis consequential error';
			17504: sMsg := 'Minimum software position limit';
			17505: sMsg := 'Maximum software position limit (axis start)';
			17135: sMsg := 'Axis is locked for motion commands because a stop command is still active';
			18000: sMsg := 'Drive hardware not ready to operate';
		ELSE
			sMsg := 'No Message Data';
		END_CASE
	END_IF
	
	GVL_machine.aErrorData[5,GVL_machine.nErrorDataRow] := sMsg;
	
	//Check if end of table was reached
	IF GVL_machine.nErrorDataRow = 23 THEN 
		GVL_machine.nErrorDataRow := 1;
	ELSE
		GVL_machine.nErrorDataRow := GVL_machine.nErrorDataRow + 1;
	END_IF

END_FUNCTION

// ---- POUs/PROGRAMS/multiControl.TcPOU
PROGRAM multiControl
VAR
	multiCtrlFrameIndex : INT; //Index used to switch frame on multiControlScreen
	
	aActionList 		: ARRAY[1..11] OF STRING := ['BRAKE OFF','BRAKE ON','DISABLE','ENABLE','HOME TO SENSOR','HOME TO TORQUE','MOVE TO POSITION','JOG','MOVE TO TORQUE','RESET','SET COUNT']; //List of usable actions found in FB_MultiMotorController.
	nActionIndex 		: INT;
	nPrevActionIndex 	: INT;
	pMotorRef1 			: POINTER TO FB_teknicMotorEC;
	pMotorRef2 			: POINTER TO FB_teknicMotorEC;
	pMotorRef3 			: POINTER TO FB_teknicMotorEC;
	pMotorRef4 			: POINTER TO FB_teknicMotorEC;
	aMotorEnabledRef 	: ARRAY[1..4] OF POINTER TO FB_teknicMotorEC; //Used to act on only motors currently enabled
	aMotorRef 			: ARRAY[1..4] OF POINTER TO FB_teknicMotorEC; // Used to update live values of motors in selection
	fRelease			: F_TRIG; 
	bReleaseTrig		: BOOL;

	// Motor Disp //
	nMotorControlIndex 		: INT; // Index used to change disp of motor controls. 0-Rotation, 1- Clamping, 2-Columns, 3-Width. 
	nPrevMotorControlIndex 	: INT; // INdex used to reset selections when frame changes 
	aDispFontColor 			: ARRAY[1..4] OF DWORD; // Used to change font color of motor display when toggled. 
	bHideDispMotor3 		: BOOL; //Used to hide or show controls for motor 3. 
	bHideDispMotor4			: BOOL;
	bHideDirection			: BOOL; //Hides direction of buttons based on selected action
	bHideSetPos				: BOOL; //Hides Set Position Entry based on selected action
	bHideSetTorq			: BOOL; //Hides Set Torque Entry based on selected action
	
	aMotorActive 	: ARRAY[1..4] OF BOOL; // Tracks user selected motors
	aMotorError 	: ARRAY[1..4] OF BOOL; // Indictates error for current action
	aMotorErrorId 	: ARRAY[1..4] OF UDINT; //Indicates error Id for current action
	aMotorDone 		: ARRAY[1..4] OF BOOL; //Indicates action is done
	aMotorInverted  : ARRAY[1..4] OF BOOL; //Indicates whether the motor is inverted
	
	sMotorDisp1 : STRING; // Used to dynamically change the title of motor 1. 
	sMotorDisp2 : STRING;
	sMotorDisp3 : STRING;
	sMotorDisp4 : STRING;
	
	// Motor Control //
	aMotorEnable 	: ARRAY[1..4] OF BOOL; //Array defining whether a motor is selected and should be used for the current action. 
	nCounter 		: INT; //Index for FOR loops.
	aMotorSpeed 	: ARRAY[1..4] OF LREAL; //Displays motors' speeds
	aMotorPos 		: ARRAY[1..4] OF LREAL; //Displays motors' positions
	aMotorTorque 	: ARRAY[1..4] OF LREAL; //Displays motors' torques
	aMotorSetPos 	: ARRAY[1..4] OF LREAL; //User set position for motors
	aMotorSetTorq 	: ARRAY[1..4] OF LREAL; //User set torque for motors
	bHomeDirection  : BOOL; // Direction of moves.
	nDirection 		: INT;	//Calculated direction based on inverted motor or not. 
	bExecute 		: BOOL; // Execute selected action 
	i : INT;
	
	// === parametersHandler Vars === //
	aStatusVar 				: ARRAY[1..12] OF BOOL; // Array containing boolean value for each status variable represented on screen. 
	aMotorSelection 		: ARRAY[1..10] OF STRING := ['LEFT ROTATION','RIGHT ROTATION','COLUMN 0','COLUMN 1','COLUMN 2','COLUMN 3','LEFT WIDTH','RIGHT WIDTH','LEFT CLAMPING','RIGHT CLAMPING']; //Drop down box to select motor to read/write
	nMotorSelectionIndex 	: INT; //Index of drop down box
	pMotorRefParam			: POINTER TO FB_teknicMotorEC;
	eParameter				: MC_AxisParameter;
	nParameterIndex			: INT; // Index of combo box for selected parameter
	fValueIn				: LREAL; // Value used to write to parameter
	fValueOut				: LREAL;// Value from read parameter. 
	bReadParam				: BOOL; // Btn used to trigger read parameter
	bWriteParam				: BOOL; // Btn used to trigger write parameter
END_VAR

CASE nMotorControlIndex OF 
	0:// Rotation Selected
		aMotorRef[1] := ADR(GVL_devices.fbLftRotationMotor);
		aMotorRef[2] := ADR(GVL_devices.fbRhtRotationMotor);
		aMotorRef[3] := 0;
		aMotorRef[4] := 0;
		IF aMotorEnable[1] THEN
			pMotorRef1 := ADR(GVL_devices.fbLftRotationMotor);
		ELSE
			pMotorRef1 := 0;
		END_IF
		IF aMotorEnable[2] THEN
			pMotorRef2 := ADR(GVL_devices.fbRhtRotationMotor);
		ELSE
			pMotorRef2 := 0;
		END_IF
		pMotorRef3 := 0;
		pMotorRef4 := 0;
	    bHideDispMotor3 := TRUE;
	    bHideDispMotor4 := TRUE;
		sMotorDisp1 := 'LEFT ROTATION';
		sMotorDisp2 := 'RIGHT ROTATION';
		sMotorDisp3 := '';
		sMotorDisp4 := '';
		
	1:// Clamping Selected
		aMotorRef[1] := ADR(GVL_devices.fbLftClampMotor);
		aMotorRef[2] := ADR(GVL_devices.fbRhtClampMotor);
		aMotorRef[3] := 0;
		aMotorRef[4] := 0;
		IF aMotorEnable[1] THEN
			pMotorRef1 := ADR(GVL_devices.fbLftClampMotor);
		ELSE
			pMotorRef1 := 0;
		END_IF
		IF aMotorEnable[2] THEN
			pMotorRef2 := ADR(GVL_devices.fbRhtClampMotor);
		ELSE
			pMotorRef2 := 0;
		END_IF
		pMotorRef3 := 0;
		pMotorRef4 := 0;
	    bHideDispMotor3 := TRUE;
	    bHideDispMotor4 := TRUE;
		sMotorDisp1 := 'LEFT CLAMPING';
		sMotorDisp2 := 'RIGHT CLAMPING';
		sMotorDisp3 := '';
		sMotorDisp4 := '';
		
	2:// Columns Selected
		aMotorRef[1] := ADR(GVL_devices.fbColumn0Motor);
		aMotorRef[2] := ADR(GVL_devices.fbColumn1Motor);
		aMotorRef[3] := ADR(GVL_devices.fbColumn2Motor);
		aMotorRef[4] := ADR(GVL_devices.fbColumn3Motor);
		
		IF aMotorEnable[1] THEN
			pMotorRef1 := ADR(GVL_devices.fbColumn0Motor);
		ELSE
			pMotorRef1 := 0;
		END_IF
		IF aMotorEnable[2] THEN
			pMotorRef2 := ADR(GVL_devices.fbColumn1Motor);
		ELSE
			pMotorRef2 := 0;
		END_IF
		IF aMotorEnable[3] THEN
			pMotorRef3 := ADR(GVL_devices.fbColumn2Motor);
		ELSE
			pMotorRef3 := 0;
		END_IF
		IF aMotorEnable[4] THEN
			pMotorRef4 := ADR(GVL_devices.fbColumn3Motor);
		ELSE
			pMotorRef4 := 0;
		END_IF
	    bHideDispMotor3 := FALSE;
	    bHideDispMotor4 := FALSE;
		sMotorDisp1 := 'COLUMN 0';
		sMotorDisp2 := 'COLUMN 1';
		sMotorDisp3 := 'COLUMN 2';
		sMotorDisp4 := 'COLUMN 3';
		
	3:// Width Selected
		aMotorRef[1] := ADR(GVL_devices.fbLftWidthMotor);
		aMotorRef[2] := ADR(GVL_devices.fbRhtWidthMotor);
		aMotorRef[3] := 0;
		aMotorRef[4] := 0;
		IF aMotorEnable[1] THEN
			pMotorRef1 := ADR(GVL_devices.fbLftWidthMotor);
		ELSE
			pMotorRef1 := 0;
		END_IF
		IF aMotorEnable[2] THEN
			pMotorRef2 := ADR(GVL_devices.fbRhtWidthMotor);
		ELSE
			pMotorRef2 := 0;
		END_IF
		pMotorRef3 := 0;
		pMotorRef4 := 0;
	    bHideDispMotor3 := TRUE;
	    bHideDispMotor4 := TRUE;
		sMotorDisp1 := 'LEFT WIDTH';
		sMotorDisp2 := 'RIGHT WIDTH';
		sMotorDisp3 := '';
		sMotorDisp4 := '';
END_CASE

aMotorEnabledRef[1] := pMotorRef1;
aMotorEnabledRef[2] := pMotorRef2;
aMotorEnabledRef[3] := pMotorRef3;
aMotorEnabledRef[4] := pMotorRef4;

// === Update Motor Displays and Position,Torque,Inverted,and Speed. === //
FOR nCounter := 1 TO 4 BY 1 DO
	IF aMotorEnable[nCounter] THEN
		aDispFontColor[nCounter] := 16#FFFFFFFF;
	ELSE
		aDispFontColor[nCounter] := 16#FF000000;
	END_IF
END_FOR

FOR nCounter := 1 TO 4 BY 1 DO
	IF aMotorRef[nCounter] <> 0 THEN
		aMotorSpeed[nCounter] := aMotorRef[nCounter]^.fbMotor.NcToPlc.ActVelo;
	END_IF
END_FOR

FOR nCounter := 1 TO 4 BY 1 DO
	IF aMotorRef[nCounter] <> 0 THEN
		aMotorPos[nCounter] := aMotorRef[nCounter]^.fbMotor.NcToPlc.ActPos;
	END_IF
END_FOR

FOR nCounter := 1 TO 4 BY 1 DO
	IF aMotorRef[nCounter] <> 0 THEN
		aMotorTorque[nCounter] := aMotorRef[nCounter]^.fbMotor.NcToPlc.ActTorque;
	END_IF
END_FOR

FOR nCounter := 1 TO 4 BY 1 DO
	IF aMotorRef[nCounter] <> 0 THEN
		aMotorInverted[nCounter] := aMotorRef[nCounter]^.isMotorInverted;
	END_IF
END_FOR

// === Clear selections and user inputs when frame changes === //
IF nPrevMotorControlIndex <> nMotorControlIndex OR nActionIndex <> nPrevActionIndex THEN
	FOR nCounter := 1 TO 4 BY 1 DO
		aMotorEnable[nCounter] := FALSE;
		aMotorSetPos[nCounter] := 0;
		aMotorSetTorq[nCounter] := 0;
		aMotorActive[nCounter] := FALSE;
		aMotorError[nCounter] := FALSE;
		aMotorErrorId[nCounter] := 0;
		aMotorDone[nCounter] := FALSE;
	END_FOR
	nPrevMotorControlIndex := nMotorControlIndex;
	nPrevActionIndex := nActionIndex;
END_IF

// === Reset Motor State Variables and FB Variables at the end of an Execute === //
fRelease(CLK:=bExecute , Q=>bReleaseTrig );
IF bReleaseTrig THEN
	FOR nCounter := 1 TO 4 BY 1 DO
		aMotorActive[nCounter] := FALSE;
		aMotorError[nCounter] := FALSE;
		aMotorErrorId[nCounter] := 0;
		aMotorDone[nCounter] := FALSE;
		IF aMotorEnabledRef[nCounter] <> 0 THEN
			aMotorEnabledRef[nCounter]^.resetMotorCommands(); 	
		END_IF
	END_FOR
END_IF

// === Default Hide controls === //
bHideSetPos	 := TRUE;
bHideSetTorq := TRUE;
bHideDirection := TRUE;

// === CASE STATEMENT to execute actions on enabled motors === //
CASE nActionIndex OF 
	0:// Brake Off
		IF bExecute THEN
			FOR i := 1 TO 4 BY 1 DO
				IF aMotorEnabledRef[i] <> 0 THEN
					IF aMotorEnabledRef[i]^.brakeOff() THEN
						aMotorDone[i] := TRUE;
					END_IF
				END_IF
			END_FOR
		END_IF
		
	1:// Brake On
		IF bExecute THEN
			FOR i := 1 TO 4 BY 1 DO
				IF aMotorEnabledRef[i] <> 0 THEN
					IF aMotorEnabledRef[i]^.brakeOn() THEN
						aMotorDone[i] := TRUE;
					END_IF
				END_IF
			END_FOR
		END_IF
		
	2:// Disable
		IF bExecute THEN
			FOR i := 1 TO 4 BY 1 DO
				IF aMotorEnabledRef[i] <> 0 THEN
					CASE aMotorEnabledRef[i]^.disable() OF
						1:// Done
							aMotorDone[i] := TRUE;
						13:// Error
							aMotorError[i] := TRUE;	
							aMotorErrorId[i] := aMotorEnabledRef[i]^.motorErrorId;
					END_CASE
				END_IF
			END_FOR
		END_IF
			
	3:// Enable
		IF bExecute THEN
			FOR i := 1 TO 4 BY 1 DO
				IF aMotorEnabledRef[i] <> 0 THEN
					CASE aMotorEnabledRef[i]^.enable() OF
						1:// Done
							aMotorDone[i] := TRUE;
						13:// Error
							aMotorError[i] := TRUE;	
							aMotorErrorId[i] := aMotorEnabledRef[i]^.motorErrorId;
					END_CASE
				END_IF
			END_FOR
		END_IF
		
	4:// homeToSensor
		IF bExecute THEN
			FOR i := 1 TO 4 BY 1 DO
				IF aMotorEnabledRef[i] <> 0 THEN
					CASE aMotorEnabledRef[i]^.homeToSensor(0) OF
						1:// Done
							aMotorDone[i] := TRUE;
						2:// Active
							aMotorActive[i] := TRUE;
						13:// Error
							aMotorError[i] := TRUE;	
							aMotorErrorId[i] := aMotorEnabledRef[i]^.motorErrorId;
					END_CASE
				END_IF
			END_FOR
		END_IF
		
	5:// homeToTorque
		bHideSetTorq := FALSE;
		IF bExecute THEN
			FOR i := 1 TO 4 BY 1 DO
				IF aMotorEnabledRef[i] <> 0 THEN
					aMotorEnabledRef[i]^.homeTorqueLimitIn := aMotorTorque[i];
					CASE aMotorEnabledRef[i]^.homeToTorque() OF
						1:// Done
							aMotorDone[i] := TRUE;
						2:// Active
							aMotorActive[i] := TRUE;
						13:// Error
							aMotorError[i] := TRUE;	
							aMotorErrorId[i] := aMotorEnabledRef[i]^.motorErrorId;
					END_CASE
				END_IF
			END_FOR
		END_IF
		
	6:// moveTo
		bHideSetPos	 := FALSE;
		IF bExecute THEN
			FOR i := 1 TO 4 BY 1 DO
				IF aMotorEnabledRef[i] <> 0 THEN
					aMotorEnabledRef[i]^.homeTorqueLimitIn := aMotorTorque[i];
					CASE aMotorEnabledRef[i]^.moveTo('NULL',aMotorSetPos[i]/25.4) OF
						1:// Done
							aMotorDone[i] := TRUE;
						2,15:// Active
							aMotorActive[i] := TRUE;
						13:// Error
							aMotorError[i] := TRUE;	
							aMotorErrorId[i] := aMotorEnabledRef[i]^.motorErrorId;
					END_CASE
				END_IF
			END_FOR
		END_IF
		
	7:// moveToJog
	bHideDirection := FALSE;
		IF bExecute THEN
			FOR i := 1 TO 4 BY 1 DO
				IF aMotorEnabledRef[i] <> 0 THEN
					IF bHomeDirection THEN
						IF aMotorEnabledRef[i]^.isMotorInverted THEN
							nDirection := 1;
						ELSE
							nDirection := 0;
						END_IF
					ELSE
						IF aMotorEnabledRef[i]^.isMotorInverted THEN
							nDirection := 0;
						ELSE
							nDirection := 1;
						END_IF
					END_IF
					CASE aMotorEnabledRef[i]^.moveToJog(nDirection) OF
						1:// Active
							aMotorActive[i] := TRUE;
						13:// Error
							aMotorError[i] := TRUE;	
							aMotorErrorId[i] := aMotorEnabledRef[i]^.motorErrorId;
					END_CASE
				END_IF
			END_FOR
		END_IF
		
	8:// moveToTorque
		bHideSetTorq	:= TRUE;
		bHideDirection 	:= FALSE;
		IF bExecute THEN
			FOR i := 1 TO 4 BY 1 DO
				IF aMotorEnabledRef[i] <> 0 THEN
					IF bHomeDirection THEN
						IF aMotorEnabledRef[i]^.isMotorInverted THEN
							nDirection := 1;
						ELSE
							nDirection := 0;
						END_IF
					ELSE
						IF aMotorEnabledRef[i]^.isMotorInverted THEN
							nDirection := 0;
						ELSE
							nDirection := 1;
						END_IF
					END_IF
					CASE aMotorEnabledRef[i]^.moveToTorque('NULL',aMotorSetTorq[i],nDirection) OF
						1:// Done
							aMotorDone[i] := TRUE;
						2:// Active
							aMotorActive[i] := TRUE;
						13:// Error
							aMotorError[i] := TRUE;	
							aMotorErrorId[i] := aMotorEnabledRef[i]^.motorErrorId;
					END_CASE
				END_IF
			END_FOR
		END_IF
		
	9:// motorReset
		IF bExecute THEN
			FOR i := 1 TO 4 BY 1 DO
				IF aMotorEnabledRef[i] <> 0 THEN
					CASE aMotorEnabledRef[i]^.reset() OF
						1:// Done
							aMotorDone[i] := TRUE;
						2:// Active
							aMotorActive[i] := TRUE;
						13:// Error
							aMotorError[i] := TRUE;	
							aMotorErrorId[i] := aMotorEnabledRef[i]^.motorErrorId;
					END_CASE
				END_IF
			END_FOR
		END_IF
		
	10:// homeSetToCount
		bHideSetPos	 := FALSE;
		IF bExecute THEN
			FOR i := 1 TO 4 BY 1 DO
				IF aMotorEnabledRef[i] <> 0 THEN
					CASE aMotorEnabledRef[i]^.homeSetToCount(aMotorSetPos[i]) OF
						1:// Done
							aMotorDone[i] := TRUE;
						2:// Active
							aMotorActive[i] := TRUE;
						13:// Error
							aMotorError[i] := TRUE;	
							aMotorErrorId[i] := aMotorEnabledRef[i]^.motorErrorId;
					END_CASE
				END_IF
			END_FOR
		END_IF
END_CASE


IF multiCtrlFrameIndex = 3 THEN
	parametersHandler();
END_IF

METHOD parametersHandler : BOOL
VAR_INPUT
END_VAR
CASE nMotorControlIndex OF 
	1://Left Rotation 
		pMotorRefParam := ADR(GVL_devices.fbLftRotationMotor);
	2://Right Rotation 
		pMotorRefParam := ADR(GVL_devices.fbRhtRotationMotor);
	3://Column 0
		pMotorRefParam := ADR(GVL_devices.fbColumn0Motor); 
	4://Column 1
		pMotorRefParam := ADR(GVL_devices.fbColumn1Motor);
	5://Column 2 
		pMotorRefParam := ADR(GVL_devices.fbColumn2Motor);
	6://Column 3
		pMotorRefParam := ADR(GVL_devices.fbColumn3Motor);
	7://Left Width
		pMotorRefParam := ADR(GVL_devices.fbLftWidthMotor);
	8://Right Width
		pMotorRefParam := ADR(GVL_devices.fbRhtWidthMotor);
	9://Left Clamp
		pMotorRefParam := ADR(GVL_devices.fbLftClampMotor);
	10://Right Clamp
		pMotorRefParam := ADR(GVL_devices.fbRhtClampMotor);
END_CASE

aStatusVar[1] := pMotorRefParam^.stMotorStatus.Error;
aStatusVar[2] := pMotorRefParam^.stMotorStatus.ErrorStop;
aStatusVar[3] := pMotorRefParam^.stMotorStatus.Disabled;
aStatusVar[4] := pMotorRefParam^.stMotorStatus.Operational;
aStatusVar[5] := pMotorRefParam^.stMotorStatus.ControlLoopClosed;
aStatusVar[6] := pMotorRefParam^.stMotorStatus.ProtectedMode;
aStatusVar[7] := pMotorRefParam^.stMotorStatus.Homed;
aStatusVar[8] := pMotorRefParam^.stMotorStatus.MotionCommandsLocked;
aStatusVar[9] := pMotorRefParam^.stMotorStatus.SoftLimitMinExceeded;
aStatusVar[10] := pMotorRefParam^.stMotorStatus.SoftLimitMaxExceeded;
aStatusVar[11] := pMotorRefParam^.stMotorStatus.DriveDeviceError;
aStatusVar[12] := pMotorRefParam^.stMotorStatus.Coupled;

eParameter := nParameterIndex;

IF bReadParam THEN
	fValueOut := pMotorRefParam^.fReadValue;
	CASE pMotorRefParam^.readRealParameter(eParameter) OF 
		1,13: bReadParam := FALSE;
			pMotorRefParam^.resetMotorCommands();
	END_CASE
END_IF

IF bWriteParam THEN
	CASE pMotorRefParam^.writeRealParameter(eParameter,fValueIn) OF 
		1,13: bWriteParam := FALSE;
			pMotorRefParam^.resetMotorCommands();
	END_CASE
END_IF
END_METHOD

END_PROGRAM

// ---- POUs/DEVICES/FB_teknicMotorEC.TcPOU
FUNCTION_BLOCK FB_teknicMotorEC
VAR
	//I/O
	bBrake			AT %Q*  : BOOL;
	bHomeSensor		AT %I*  : BOOL;
	bClampSensor 	AT %I*  : BOOL;
	bTempCylinder   AT %Q*  : BOOL; //TEMP CODE UNTIL CYLINDER IS CHANGED BACK TO BALL SCREW.
	fHeightDisp				: REAL;
	
	//Init
	bMotorInverted : BOOL;
	bMotorDisables : BOOL;
	
	fMoveAccl 		: LREAL := 50;
	fMoveDcl 		: LREAL := 50;
	fMoveVelocity 	: LREAL;
	
	torqueVelocity		: LREAL;
	torqueAcceleration	: LREAL;
	torqueDeceleration	: LREAL;
	
	homeVelocity		: LREAL;
	homeSetPosition		: LREAL;
	homeTorqueLimit		: LREAL;
	
	jogTorque			: LREAL;
	
	bHasHomeSensor		: BOOL;
	
	//State Var
	nMoveState 				: INT;
	nMoveStateTorque		: INT;
	nHomeState				: INT;
	nInitState 				: INT;
	nResetState 			: INT;
	estopState 				: INT := 0; // 0 = Idle, 3 = GearOut, 2 = Stop, 1 = Done
	stopState				: INT;
	
	bIdle 					: BOOL;
	bIdleEnabled 			: BOOL;
	bIdleDisabled 			: BOOL;
	
	fMinHeight				: REAL;
	fMaxHeight 				: REAL := 115;
	fPrevHeight				: REAL;
	bSensorWarning			: BOOL;
	fHeight					: REAL;
	nMoveUpCount			: INT;
	nMoveDownCount			: INT;

	stError : ST_errorRef;
	
	// Timer to turn brake on if motor is left holding carriage for so long;
	fbBrakeTimer 	: TON;
	bIn				: BOOL;
	tPt				: TIME := T#1M;
	bQ				: BOOL;
	tEt				: TIME;
	
	/////////// EC Motor //////////////////////////////////
	fbMotor : axis_REF;
	
	//Power
	fbMotorPower	: MC_Power;
	stMotorPowerOut : ST_McOutputs;
	
	//Reset
	fbMotorReset 	: MC_RESET;
	stMotorResetOut : ST_McOutputs;

	//Halt
	fbMotorHalt 	: MC_HALT;
	stMotorHaltOut 	: ST_McOutputs;
	
	//Velocity Jog
	fbMotorJog 		: MC_JOG;
	stMotorJogOut 	: ST_McOutputs;
	eJogMode 		: E_JogMode;
	nJogModeSelect 	: INT := 2;
	

	//Homing
	fbMotorHome		: MC_Home;
	stHomingOptions : ST_HomingOptions;
	stMotorHomeOut 	: ST_McOutputs;
	bDummyHomingCam : BOOL;
	stHomingMode 	: MC_HomingMode;
	bCheckhomeSensor: BOOL;
	bMotorHomeStatus: BOOL;
	bHomeSensorTriggered : BOOL;
	fbFreeSensorTimer : TON;
	
	//Mode
	fbMotorWriteMode	: MC_WriteDriveOperationMode;
	stMotorWriteModeOut : ST_McOutputs;
	fbMotorReadMode		: MC_ReadDriveOperationMode;
	stMotorReadModeOut 	: ST_McOutputs;
	stOpModeMotor 		: E_DriveOperationMode;
	stOpModeMotorInt	: DINT;
	stWriteMode 		: E_DriveOperationMode;
	nWriteModeSelect 	: DINT := 0;
	fbReadBoolParam		: MC_readParameter;
	fbReadRealParam		: MC_readParameter;
	stReadParamOut 		: ST_mcOutputs;
	eParameter 			: MC_AxisParameter; //Parameter to read or write. https://infosys.beckhoff.com/english.php?content=../content/1033/tcplclib_tc2_mc2/70069259.html&id=
	fReadValue 			: LREAL; // Return value when MC_AxisParameter is of type REAL
	bReadValue 			: LREAL; // Return value when MC_AxisParameter is of type BOOL
	fbWriteRealParam	: MC_WriteParameter;
	fbWriteBoolParam	: MC_WriteParameter;
	stWriteParameterOut : ST_mcOutputs;
	fWriteValue 		: LREAL; // Write value when MC_AxisParameter is of type REAL
	bWriteValue			: BOOL; // Write value when MC_AxisParameter is of type BOOL
	
	//Move Absolute
	fbMotorMoveAbsolute		: MC_MoveAbsolute;
	stMotorMoveAbsoluteOut 	: ST_mcOutputs;
	bChangePosition 		: BOOL;
	fPosition 				: LREAL := 300;
	fStartPos				: LREAL;
	fHalfwayPos				: LREAL;
	
	//Move Relative
	fbMotorMoveRelative		: MC_MoveRelative;
	stMotorMoveRelativeOut 	: ST_McOutputs;
	
	//Move Velocity
	fbMotorMoveVelocity		: MC_MoveVelocity;
	stMotorMoveVelocityOut	: ST_mcOutputs;
	fVel 					: LREAL := 100;
	stDirection 			: MC_Direction;
	stDirectionSelect 		: INT := 1;

	// Stop
	fbMotorStop		: MC_Stop;
	stMotorStopOut 	: ST_mcOutputs;
	bExectuteStop 	: BOOL;
	bStopDone 		: BOOL;
	bStopBtn 		: BOOL;
	
	//Torque
	fbMotorTorque		: FB_moveToTorque;
	stMotorTorqueOut 	: ST_mcOutputs;
	fTorque 			: LREAL := 2;
	torqueDirection		: INT;
	torqueTime			: TIME := T#100MS;

	//Gear Coupling
	fbMotorGearIn : MC_GearIn;
	fbMotorGearOut: MC_GearOut;
	stMotorGearInOut : ST_McOutputs;
	stMotorGearOutOut: ST_McOutputs;
	refMasterAxis : axis_REF;
	
	//Status
	fbMotorReadStatus 		: MC_ReadStatus;
	stMotorStatus 			: ST_AxisStatus;
	stMotorReadStatusOut 	: ST_mcOutputs;
	
	//Set Position
	fbMotorSetPosition			: MC_SetPosition;
	stMotorSetPositionOut 		: ST_mcOutputs;
	stMotorSetPositionOption 	: ST_SetPositionOptions;

	fbMotorWriteParameter	: MC_WriteParameter;
	stMotorWriteOut 		: ST_mcOutputs;
	
	sModeDisp 		: STRING;
	fbReadModeTimer	: TON;
	
	//Home to Torque	
	fbHomeToTorque		: FB_homeToTorque;
	stHomeToTorqueOut 	: ST_mcOutputs;
	direction			: INT; // 0- PositiveDirection, 1- NegativeDirection
	homeTimeLimit		: TIME := T#2M;
	homeBackOffPos		: LREAL := 10;
	
	//Home to Sensor Custom 
	fbHomeToSensorCustom : FB_homeToSensorCustom;
	stHomeToSensorCustomOut : ST_McOutputs;
	
	bUsingStopReset: BOOL;
END_VAR

(* Behavior of this motor setup is a steady state of disabling the motor when no command is being executed. This setup is best with motors that have a brake
connected to the PLC or motors connected to systems where the system can remain still without assistance from the motor. 
*)
fbBrakeTimer(IN:= bIn, PT:= tPt, Q=> bQ, ET=> tEt);
IF GVL_machine.bMotorsInitialized AND nResetState = 0 THEN
	//bUsingStopReset := FALSE;
	IF bIdleDisabled THEN 
		bIn := TRUE;
	ELSE
		bIn := FALSE;
	END_IF
	
	IF bQ THEN
		IF fbMotor.status.HasJob THEN 
			bIn := FALSE;
		ELSE
			stop();
			brakeOn();
		END_IF
		
	END_IF
	
	(*IF bIdle THEN
		bIdleDisabled R= bIdle;
		bIdleEnabled S= SEL(stop() = 1,FALSE,TRUE);
	ELSE
		bIdleEnabled R= NOT bIdle;
		bIdleDisabled S= SEL(removeStop() = 1,FALSE,TRUE);
	END_IF*)
	IF bIdle THEN
		bIdleDisabled R= bIdle;
		IF (fbMotor.Status.HasBeenStopped OR fbMotor.Status.StandStill) AND bIdleEnabled THEN
			stopState := 0;
			fbMotorStop.Execute := FALSE;
		ELSE
			bIdleEnabled := SEL(stop() = 1,FALSE,TRUE);
			//bUsingStopReset := TRUE;
		END_IF
	ELSE
		bIdleEnabled R= NOT bIdle;
		IF (fbMotor.Status.HasBeenStopped OR fbMotor.Status.StandStill) AND NOT bIdleDisabled THEN
			bIdleDisabled := SEL(removeStop() = 1,FALSE,TRUE);
		ELSE
			stopState := 0;
		END_IF
	END_IF
END_IF

	
actPower();
actHome();
actMode();
actStop();
actMove();
actTorque();
actCouple();
actStatus();


fbMotor();
fbMotorJog.JogForward := FALSE;
fbMotorJog.JogBackwards := FALSE;

ACTION actCouple:
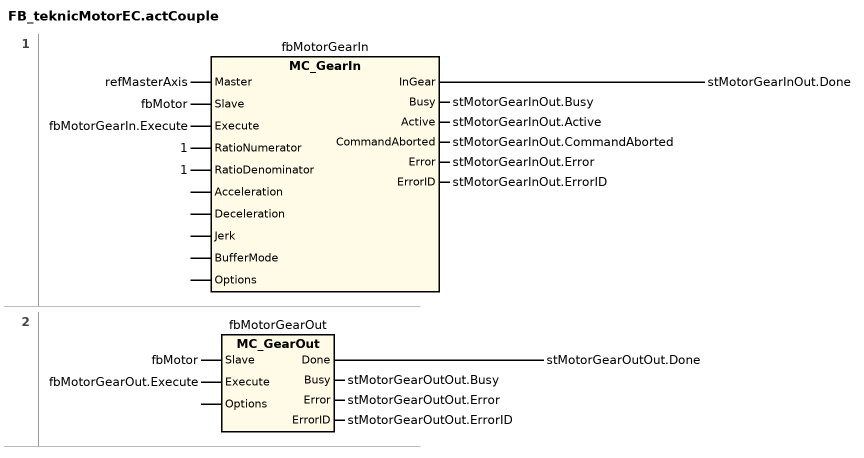
// NETWORK 1
fbMotorGearIn(
    Master := refMasterAxis,
    Slave := fbMotor,
    Execute := fbMotorGearIn.Execute,
    RatioNumerator := 1,
    RatioDenominator := 1,
    Busy => stMotorGearInOut.Busy,
    Active => stMotorGearInOut.Active,
    CommandAborted => stMotorGearInOut.CommandAborted,
    Error => stMotorGearInOut.Error,
    ErrorID => stMotorGearInOut.ErrorID); // MC_GearIn
stMotorGearInOut.Done := fbMotorGearIn.InGear;

// NETWORK 2
fbMotorGearOut(
    Slave := fbMotor,
    Execute := fbMotorGearOut.Execute,
    Busy => stMotorGearOutOut.Busy,
    Error => stMotorGearOutOut.Error,
    ErrorID => stMotorGearOutOut.ErrorID); // MC_GearOut
stMotorGearOutOut.Done := fbMotorGearOut.Done;
END_ACTION

ACTION actHome:
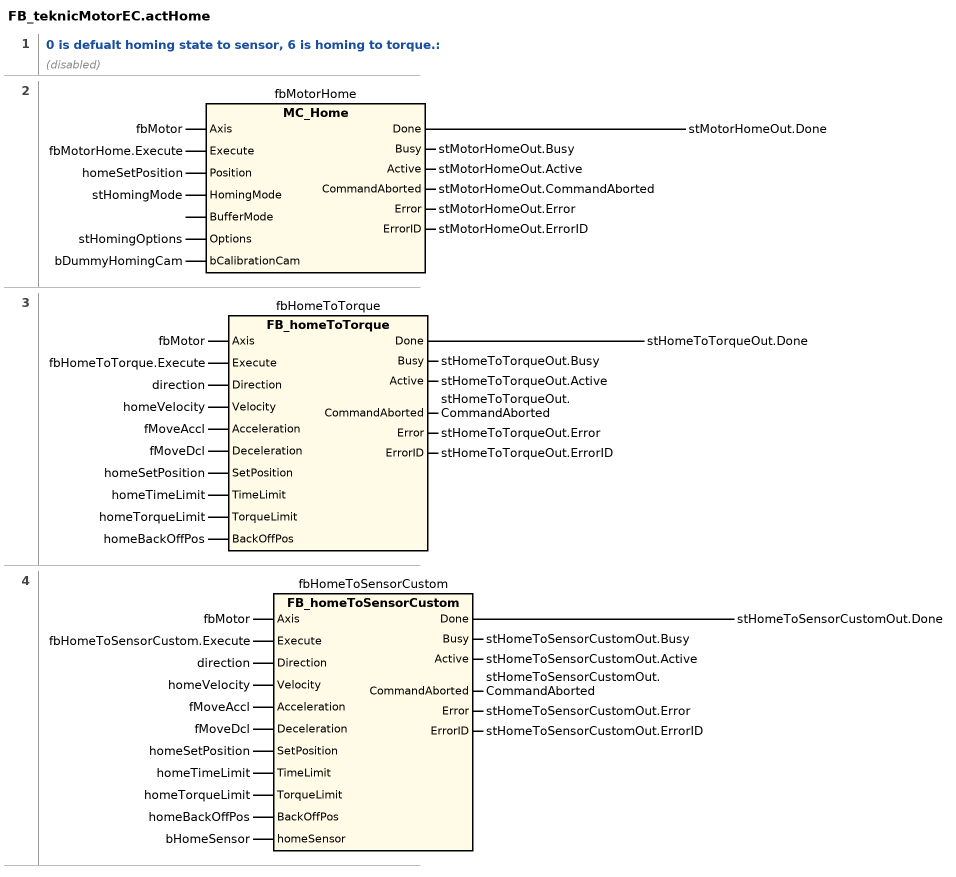
// NETWORK 1 (disabled)
// label: 0 is defualt homing state to sensor, 6 is homing to torque.

// NETWORK 2
fbMotorHome(
    Axis := fbMotor,
    Execute := fbMotorHome.Execute,
    Position := homeSetPosition,
    HomingMode := stHomingMode,
    Options := stHomingOptions,
    bCalibrationCam := bDummyHomingCam,
    Busy => stMotorHomeOut.Busy,
    Active => stMotorHomeOut.Active,
    CommandAborted => stMotorHomeOut.CommandAborted,
    Error => stMotorHomeOut.Error,
    ErrorID => stMotorHomeOut.ErrorID); // MC_Home
stMotorHomeOut.Done := fbMotorHome.Done;

// NETWORK 3
fbHomeToTorque(
    Axis := fbMotor,
    Execute := fbHomeToTorque.Execute,
    Direction := direction,
    Velocity := homeVelocity,
    Acceleration := fMoveAccl,
    Deceleration := fMoveDcl,
    SetPosition := homeSetPosition,
    TimeLimit := homeTimeLimit,
    TorqueLimit := homeTorqueLimit,
    BackOffPos := homeBackOffPos,
    Busy => stHomeToTorqueOut.Busy,
    Active => stHomeToTorqueOut.Active,
    CommandAborted => stHomeToTorqueOut.CommandAborted,
    Error => stHomeToTorqueOut.Error,
    ErrorID => stHomeToTorqueOut.ErrorID); // FB_homeToTorque
stHomeToTorqueOut.Done := fbHomeToTorque.Done;

// NETWORK 4
fbHomeToSensorCustom(
    Axis := fbMotor,
    Execute := fbHomeToSensorCustom.Execute,
    Direction := direction,
    Velocity := homeVelocity,
    Acceleration := fMoveAccl,
    Deceleration := fMoveDcl,
    SetPosition := homeSetPosition,
    TimeLimit := homeTimeLimit,
    TorqueLimit := homeTorqueLimit,
    BackOffPos := homeBackOffPos,
    homeSensor := bHomeSensor,
    Busy => stHomeToSensorCustomOut.Busy,
    Active => stHomeToSensorCustomOut.Active,
    CommandAborted => stHomeToSensorCustomOut.CommandAborted,
    Error => stHomeToSensorCustomOut.Error,
    ErrorID => stHomeToSensorCustomOut.ErrorID); // FB_homeToSensorCustom
stHomeToSensorCustomOut.Done := fbHomeToSensorCustom.Done;
END_ACTION

ACTION actMode:
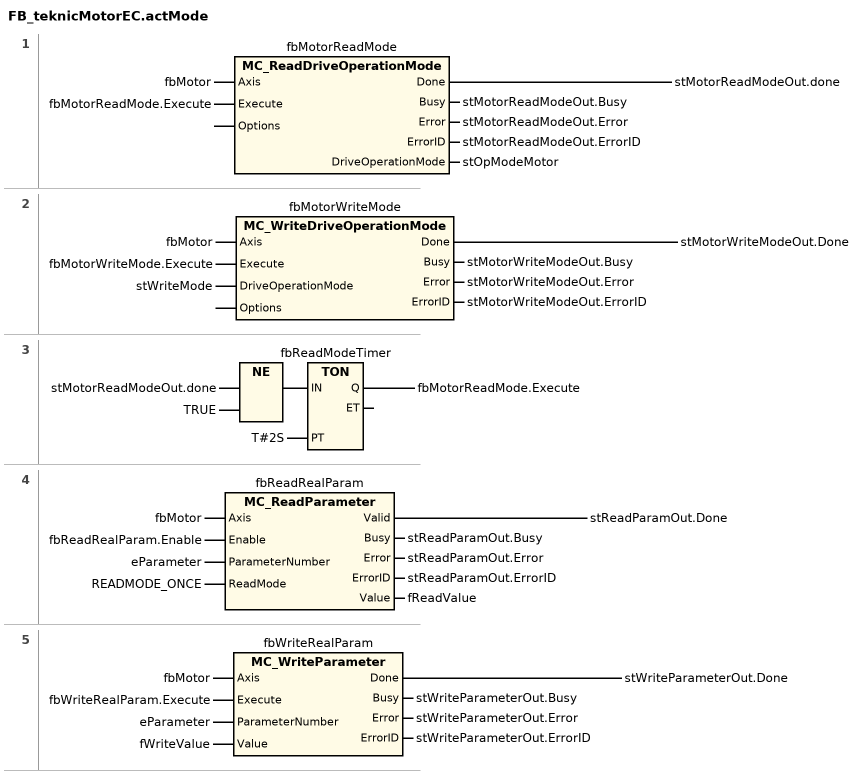
// NETWORK 1
fbMotorReadMode(
    Axis := fbMotor,
    Execute := fbMotorReadMode.Execute,
    Busy => stMotorReadModeOut.Busy,
    Error => stMotorReadModeOut.Error,
    ErrorID => stMotorReadModeOut.ErrorID,
    DriveOperationMode => stOpModeMotor); // MC_ReadDriveOperationMode
stMotorReadModeOut.done := fbMotorReadMode.Done;

// NETWORK 2
fbMotorWriteMode(
    Axis := fbMotor,
    Execute := fbMotorWriteMode.Execute,
    DriveOperationMode := stWriteMode,
    Busy => stMotorWriteModeOut.Busy,
    Error => stMotorWriteModeOut.Error,
    ErrorID => stMotorWriteModeOut.ErrorID); // MC_WriteDriveOperationMode
stMotorWriteModeOut.Done := fbMotorWriteMode.Done;

// NETWORK 3
fbReadModeTimer(IN := stMotorReadModeOut.done <> TRUE, PT := T#2S); // TON
fbMotorReadMode.Execute := fbReadModeTimer.Q;

// NETWORK 4
fbReadRealParam(
    Axis := fbMotor,
    Enable := fbReadRealParam.Enable,
    ParameterNumber := eParameter,
    ReadMode := READMODE_ONCE,
    Busy => stReadParamOut.Busy,
    Error => stReadParamOut.Error,
    ErrorID => stReadParamOut.ErrorID,
    Value => fReadValue); // MC_ReadParameter
stReadParamOut.Done := fbReadRealParam.Valid;

// NETWORK 5
fbWriteRealParam(
    Axis := fbMotor,
    Execute := fbWriteRealParam.Execute,
    ParameterNumber := eParameter,
    Value := fWriteValue,
    Busy => stWriteParameterOut.Busy,
    Error => stWriteParameterOut.Error,
    ErrorID => stWriteParameterOut.ErrorID); // MC_WriteParameter
stWriteParameterOut.Done := fbWriteRealParam.Done;
END_ACTION

ACTION actMove:
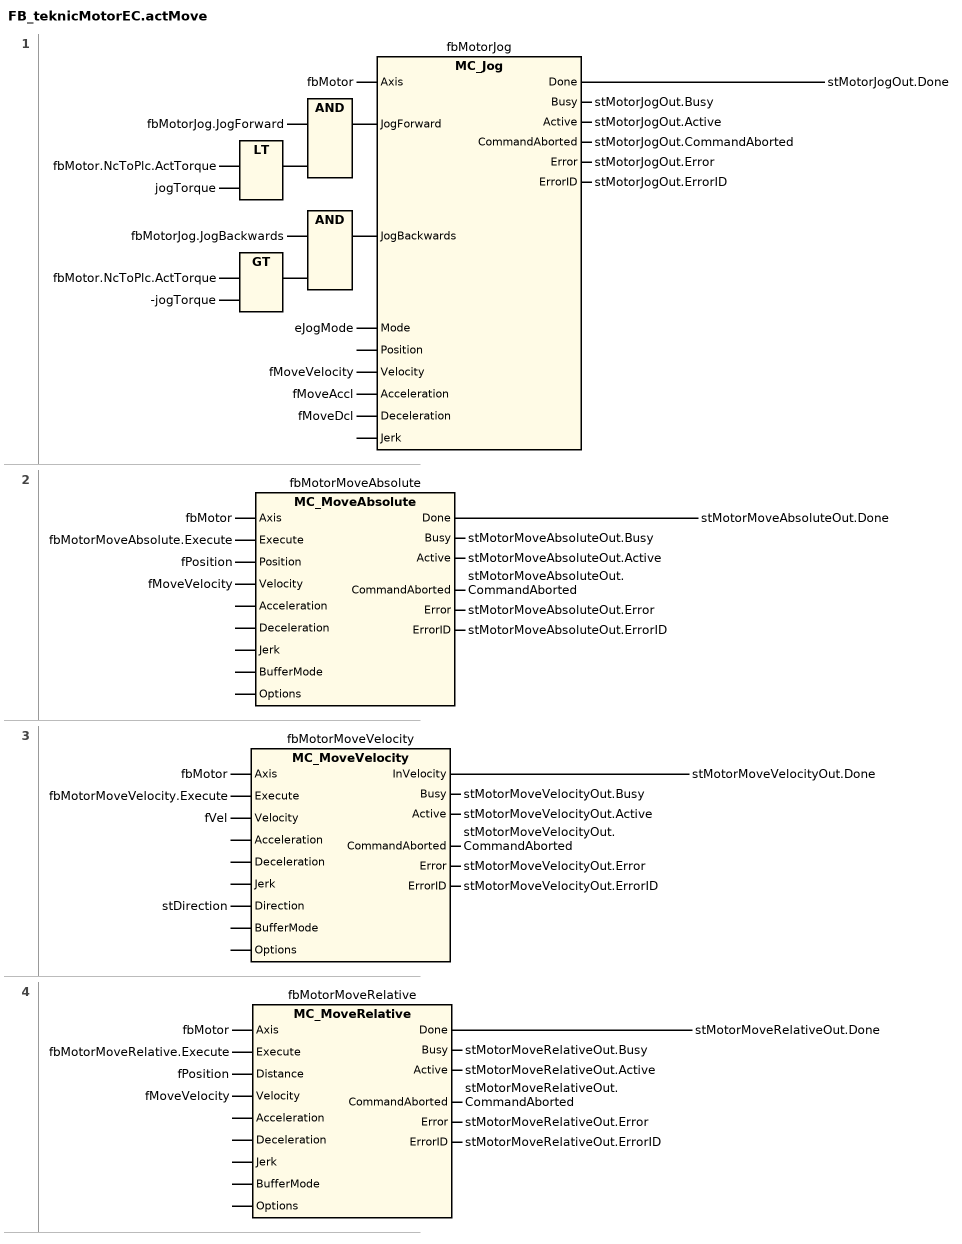
// NETWORK 1
fbMotorJog(
    Axis := fbMotor,
    JogForward := fbMotorJog.JogForward AND fbMotor.NcToPlc.ActTorque < jogTorque,
    JogBackwards := fbMotorJog.JogBackwards AND fbMotor.NcToPlc.ActTorque > (-jogTorque),
    Mode := eJogMode,
    Velocity := fMoveVelocity,
    Acceleration := fMoveAccl,
    Deceleration := fMoveDcl,
    Busy => stMotorJogOut.Busy,
    Active => stMotorJogOut.Active,
    CommandAborted => stMotorJogOut.CommandAborted,
    Error => stMotorJogOut.Error,
    ErrorID => stMotorJogOut.ErrorID); // MC_Jog
stMotorJogOut.Done := fbMotorJog.Done;

// NETWORK 2
fbMotorMoveAbsolute(
    Axis := fbMotor,
    Execute := fbMotorMoveAbsolute.Execute,
    Position := fPosition,
    Velocity := fMoveVelocity,
    Busy => stMotorMoveAbsoluteOut.Busy,
    Active => stMotorMoveAbsoluteOut.Active,
    CommandAborted => stMotorMoveAbsoluteOut.CommandAborted,
    Error => stMotorMoveAbsoluteOut.Error,
    ErrorID => stMotorMoveAbsoluteOut.ErrorID); // MC_MoveAbsolute
stMotorMoveAbsoluteOut.Done := fbMotorMoveAbsolute.Done;

// NETWORK 3
fbMotorMoveVelocity(
    Axis := fbMotor,
    Execute := fbMotorMoveVelocity.Execute,
    Velocity := fVel,
    Direction := stDirection,
    Busy => stMotorMoveVelocityOut.Busy,
    Active => stMotorMoveVelocityOut.Active,
    CommandAborted => stMotorMoveVelocityOut.CommandAborted,
    Error => stMotorMoveVelocityOut.Error,
    ErrorID => stMotorMoveVelocityOut.ErrorID); // MC_MoveVelocity
stMotorMoveVelocityOut.Done := fbMotorMoveVelocity.InVelocity;

// NETWORK 4
fbMotorMoveRelative(
    Axis := fbMotor,
    Execute := fbMotorMoveRelative.Execute,
    Distance := fPosition,
    Velocity := fMoveVelocity,
    Busy => stMotorMoveRelativeOut.Busy,
    Active => stMotorMoveRelativeOut.Active,
    CommandAborted => stMotorMoveRelativeOut.CommandAborted,
    Error => stMotorMoveRelativeOut.Error,
    ErrorID => stMotorMoveRelativeOut.ErrorID); // MC_MoveRelative
stMotorMoveRelativeOut.Done := fbMotorMoveRelative.Done;
END_ACTION

ACTION actPower:
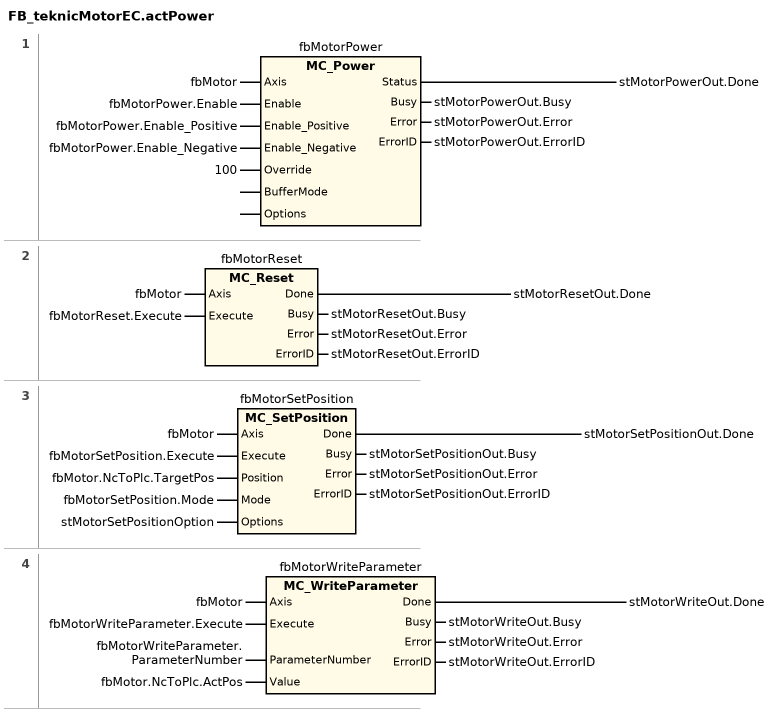
// NETWORK 1
fbMotorPower(
    Axis := fbMotor,
    Enable := fbMotorPower.Enable,
    Enable_Positive := fbMotorPower.Enable_Positive,
    Enable_Negative := fbMotorPower.Enable_Negative,
    Override := 100,
    Busy => stMotorPowerOut.Busy,
    Error => stMotorPowerOut.Error,
    ErrorID => stMotorPowerOut.ErrorID); // MC_Power
stMotorPowerOut.Done := fbMotorPower.Status;

// NETWORK 2
fbMotorReset(
    Axis := fbMotor,
    Execute := fbMotorReset.Execute,
    Busy => stMotorResetOut.Busy,
    Error => stMotorResetOut.Error,
    ErrorID => stMotorResetOut.ErrorID); // MC_Reset
stMotorResetOut.Done := fbMotorReset.Done;

// NETWORK 3
fbMotorSetPosition(
    Axis := fbMotor,
    Execute := fbMotorSetPosition.Execute,
    Position := fbMotor.NcToPlc.TargetPos,
    Mode := fbMotorSetPosition.Mode,
    Options := stMotorSetPositionOption,
    Busy => stMotorSetPositionOut.Busy,
    Error => stMotorSetPositionOut.Error,
    ErrorID => stMotorSetPositionOut.ErrorID); // MC_SetPosition
stMotorSetPositionOut.Done := fbMotorSetPosition.Done;

// NETWORK 4
fbMotorWriteParameter(
    Axis := fbMotor,
    Execute := fbMotorWriteParameter.Execute,
    ParameterNumber := fbMotorWriteParameter.ParameterNumber,
    Value := fbMotor.NcToPlc.ActPos,
    Busy => stMotorWriteOut.Busy,
    Error => stMotorWriteOut.Error,
    ErrorID => stMotorWriteOut.ErrorID); // MC_WriteParameter
stMotorWriteOut.Done := fbMotorWriteParameter.Done;
END_ACTION

ACTION actStatus:
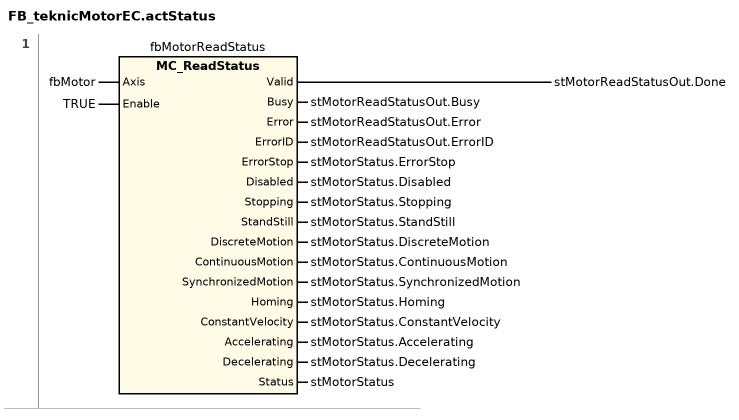
// NETWORK 1
fbMotorReadStatus(
    Axis := fbMotor,
    Enable := TRUE,
    Busy => stMotorReadStatusOut.Busy,
    Error => stMotorReadStatusOut.Error,
    ErrorID => stMotorReadStatusOut.ErrorID,
    ErrorStop => stMotorStatus.ErrorStop,
    Disabled => stMotorStatus.Disabled,
    Stopping => stMotorStatus.Stopping,
    StandStill => stMotorStatus.StandStill,
    DiscreteMotion => stMotorStatus.DiscreteMotion,
    ContinuousMotion => stMotorStatus.ContinuousMotion,
    SynchronizedMotion => stMotorStatus.SynchronizedMotion,
    Homing => stMotorStatus.Homing,
    ConstantVelocity => stMotorStatus.ConstantVelocity,
    Accelerating => stMotorStatus.Accelerating,
    Decelerating => stMotorStatus.Decelerating,
    Status => stMotorStatus); // MC_ReadStatus
stMotorReadStatusOut.Done := fbMotorReadStatus.Valid;
END_ACTION

ACTION actStop:
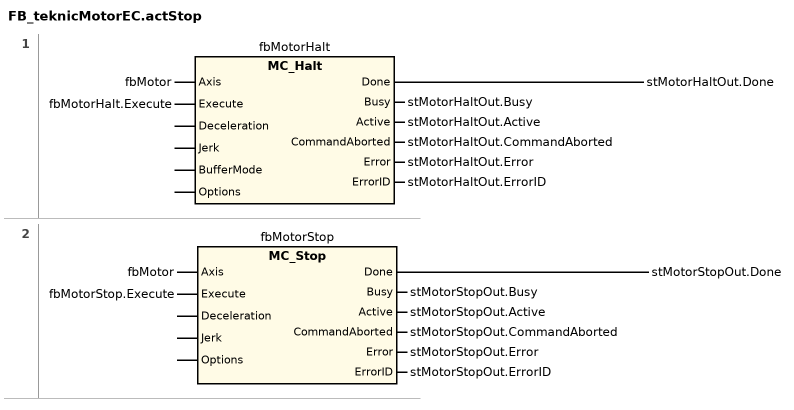
// NETWORK 1
fbMotorHalt(
    Axis := fbMotor,
    Execute := fbMotorHalt.Execute,
    Busy => stMotorHaltOut.Busy,
    Active => stMotorHaltOut.Active,
    CommandAborted => stMotorHaltOut.CommandAborted,
    Error => stMotorHaltOut.Error,
    ErrorID => stMotorHaltOut.ErrorID); // MC_Halt
stMotorHaltOut.Done := fbMotorHalt.Done;

// NETWORK 2
fbMotorStop(
    Axis := fbMotor,
    Execute := fbMotorStop.Execute,
    Busy => stMotorStopOut.Busy,
    Active => stMotorStopOut.Active,
    CommandAborted => stMotorStopOut.CommandAborted,
    Error => stMotorStopOut.Error,
    ErrorID => stMotorStopOut.ErrorID); // MC_Stop
stMotorStopOut.Done := fbMotorStop.Done;
END_ACTION

ACTION actTorque:
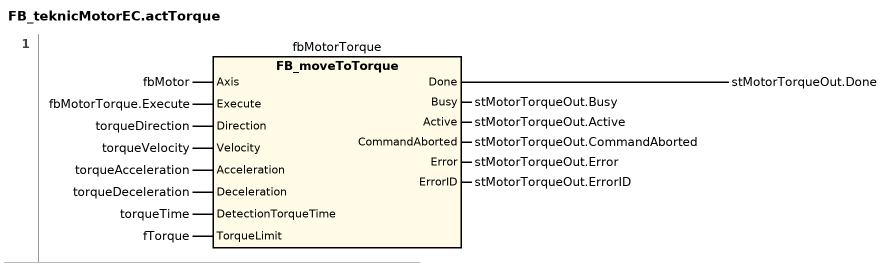
// NETWORK 1
fbMotorTorque(
    Axis := fbMotor,
    Execute := fbMotorTorque.Execute,
    Direction := torqueDirection,
    Velocity := torqueVelocity,
    Acceleration := torqueAcceleration,
    Deceleration := torqueDeceleration,
    DetectionTorqueTime := torqueTime,
    TorqueLimit := fTorque,
    Busy => stMotorTorqueOut.Busy,
    Active => stMotorTorqueOut.Active,
    CommandAborted => stMotorTorqueOut.CommandAborted,
    Error => stMotorTorqueOut.Error,
    ErrorID => stMotorTorqueOut.ErrorID); // FB_moveToTorque
stMotorTorqueOut.Done := fbMotorTorque.Done;
END_ACTION

METHOD brakeOff : BOOL
VAR_INPUT
END_VAR
bBrake := TRUE;
END_METHOD

METHOD brakeOn : BOOL
VAR_INPUT
END_VAR
bBrake := FALSE;
END_METHOD

PROPERTY camSensor : BOOL
GET
camSensor := bDummyHomingCam;
END_GET
END_PROPERTY

METHOD checkOutputs : INT
VAR_INPUT
	stRefFB : REFERENCE TO ST_McOutputs;
END_VAR
checkOutputs := 0;
IF stRefFB.Error THEN
	checkOutputs := 13;
ELSIF stRefFB.Done THEN
	checkOutputs := 1;	
ELSIF stRefFB.Active THEN
	checkOutputs := 2;
ELSIF stRefFB.Busy THEN 
	checkOutputs := 3;
ELSIF stRefFB.CommandAborted THEN
	checkOutputs := 4;
END_IF
END_METHOD

METHOD coupleToAxis : INT
VAR_INPUT
	refMasterAxisIn : REFERENCE TO axis_REF; // Master axis to couple current axis too. 
END_VAR
coupleToAxis := 0;
refMasterAxis := refMasterAxisIn;
bIdle := FALSE;
motorIdle := FALSE;
IF bIdleDisabled THEN
	fbMotorGearIn.Execute := TRUE;
	CASE checkOutputs(stMotorGearInOut) OF 
		1:// Done
			fbMotorGearIn.Execute := FALSE;
			coupleToAxis := 1;
		2:// Active	
		3:// Busy
		4:// Command Aborted
		13:// Error
			stError.errorState := MCGEARIN;
			stError.errorLoc := 'Height Motor coupleToAxis';
			setError(stMotorGearInOut);
			coupleToAxis := 13;
	END_CASE 
ELSE
	fbMotorGearIn.Execute := FALSE;
END_IF
END_METHOD

METHOD decoupleAxis : INT
VAR_INPUT
END_VAR
decoupleAxis := 0;
fbMotorGearIn.Execute := FALSE;
fbMotorGearOut.Execute := TRUE;
CASE checkOutputs(stMotorGearOutOut) OF 
	1:// Done
		fbMotorGearOut.Execute := FALSE;
		decoupleAxis := 1;
	2:// Active	
	3:// Busy
	4:// Command Aborted
	13:// Error
		stError.errorState := MCGEAROUT;
		stError.errorLoc := 'Height Motor decoupleAxis';
		setError(stMotorGearOutOut);
		decoupleAxis := 13;
END_CASE 

stop();
END_METHOD

METHOD disable : INT
VAR_INPUT
END_VAR
disable := 0;
fbMotorPower.Enable := FALSE;
fbMotorPower.Enable_Negative := FALSE;
fbMotorPower.Enable_Positive := FALSE;

IF NOT stMotorPowerOut.Busy AND NOT stMotorPowerOut.Active THEN 
	brakeOn();
	fbMotorPower.Enable := FALSE;
	disable := 1;
ELSIF stMotorPowerOut.Error THEN
	stError.errorState := MCPOWER;
	stError.errorLoc :=  'teknicMotorHeight_disable';
	setError(stMotorPowerOut);
	disable := 13;
END_IF
END_METHOD

PROPERTY distance : REAL;
GET
distance := fbMotor.NcToPlc.ActPos;
END_GET
END_PROPERTY

METHOD enable : INT //1: done, 2: Busy , 13: error
VAR_INPUT
END_VAR
enable := 0;
fbMotorPower.Enable := TRUE;
fbMotorPower.Enable_Negative := TRUE;
fbMotorPower.Enable_Positive := TRUE;

CASE checkOutputs(stMotorPowerOut) OF 
	13:// Error
		enable := 13;
	3:// Busy
		enable := 2;
	1:// Done
		enable := 1;
END_CASE
END_METHOD

METHOD estop : INT
VAR_INPUT
END_VAR
(*
estop := 0;
IF fbMotor.Status.Coupled THEN
	decoupleAxis();
ELSE 
	fbMotorStop.Execute := TRUE;
	
	CASE checkOutputs(stMotorStopOut) OF 
		1:// Done
			brakeOn();
			fbMotorPower.Enable := FALSE;
			estop := 1;
		2:// Active
		3:// Busy
		4:// Command Aborted
		13:// Error
			stError.errorState := MCSTOP;
			stError.errorLoc := 'Height Motor Stop';
			setError(stMotorStopOut);
			estop := 13;
	END_CASE
END_IF
*)
estop := 0;

CASE estopState OF
    0: // Start estop
        IF fbMotor.Status.Coupled THEN
            decoupleAxis();
            estopState := 1;
        ELSE
            fbMotorStop.Execute := TRUE;
            estopState := 2;
        END_IF

    1: // Wait for GearOut.Done
        decoupleAxis();
        IF decoupleAxis() = 1 THEN
            fbMotorStop.Execute := TRUE;
            estopState := 2;
        ELSIF decoupleAxis() = 13 THEN
            estop := 13;
            estopState := 0;
        END_IF

    2: // Wait for MC_Stop.Done
        CASE checkOutputs(stMotorStopOut) OF 
            1: // Done
                brakeOn();
                fbMotorPower.Enable := FALSE;
                estop := 1;
                estopState := 0;
            2: // Active
            3: // Busy
            4: // Command Aborted
            13: // Error
                stError.errorState := MCSTOP;
                stError.errorLoc := 'Height Motor Stop';
                setError(stMotorStopOut);
                estop := 13;
                estopState := 0;
        END_CASE

    3: // Done
        // estop complete — remain here or reset estopState externally
END_CASE
END_METHOD

METHOD homeSetToCount : INT //0:Not done, 1:done, 13: error
VAR_INPUT
	count : LREAL; // Homing that sets count to motor without movement of motor. 
END_VAR
bIdle := FALSE;
IF bIdleDisabled THEN
		//Force motor calibration without move.
		bMotorHomeStatus 	:= TRUE;
		homeSetPosition		:= count;
		stHomingMode 		:= MC_Direct;
		
		fbMotorHome.Execute := TRUE;
		actHome();
		CASE checkOutputs(stMotorHomeOut) OF 
			1:// Done
				fbMotorHome.Execute := FALSE;
				homeSetToCount := 1; 
			2:// Active
				homeSetToCount := 2;
			3:// Busy
			4:// Command Aborted
			13:// Error
				stError.errorState := MCHOME;
				stError.errorLoc := 'homeToZero';
				setError(stMotorHomeOut);
				homeSetToCount := 13;
		END_CASE
	
END_IF
END_METHOD

PROPERTY homeTorqueLimitIn : LREAL
SET
homeTorqueLimit := homeTorqueLimitIn;
END_SET
END_PROPERTY

METHOD homeToSensor : INT //0:Not done, 1:done, 2:Active, 13: error
VAR_INPUT
	stHomingSelect : INT := 0; // 0: Default Homing, 1: Sets the axis position directly to Position without executing a movement --CHANGE fHomingPos to desired Count.
END_VAR

(* Need to figure out torque value for homing.
Need to determine which direction of travel to enable*)
////////////////////////////////////////////////////////////
bIdle := FALSE;
IF bIdleDisabled THEN
	IF NOT bMotorHomeStatus THEN
		fbFreeSensorTimer(PT:=T#1S);
		IF NOT bCheckhomeSensor THEN
 			IF bHomeSensor THEN 
				//Force motor calibration without move.
				bMotorHomeStatus := TRUE;
				stHomingSelect := 2;
				CASE stHomingSelect OF 
					0: stHomingMode := MC_DefaultHoming;
					1: stHomingMode := MC_Direct;
					2: stHomingMode := MC_ForceCalibration;
					3: stHomingMode := MC_ResetCalibration;
				END_CASE
				fbMotorHome.Execute := TRUE;
				actHome();
				CASE checkOutputs(stMotorHomeOut) OF 
					1:// Done
						fbMotorHome.Execute := FALSE;
						homeToSensor := 1; 
					2:// Active
						homeToSensor := 2;
					3:// Busy
					4:// Command Aborted
					13:// Error
						stError.errorState := MCHOME;
						stError.errorLoc := 'homeToSensor_actual';
						setError(stMotorHomeOut);
						homeToSensor := 13;
				END_CASE
			END_IF
			bCheckHomeSensor := TRUE;
		ELSE
			homeToSensor := 0;
			//Homing Mode 
			CASE stHomingSelect OF 
				0: stHomingMode := MC_DefaultHoming;
				1: stHomingMode := MC_Direct;
				2: stHomingMode := MC_ForceCalibration;
				3: stHomingMode := MC_ResetCalibration;
			END_CASE
			fbMotorHome.Execute := TRUE;
			CASE checkOutputs(stMotorHomeOut) OF 
				1:// Done
					fbMotorHome.Execute := FALSE;
					homeToSensor := 1; 
				2:// Active
					homeToSensor := 2;
				3:// Busy
				4:// Command Aborted
				13:// Error
					stError.errorState := MCHOME;
					stError.errorLoc := 'homeToSensor_actual';
					setError(stMotorHomeOut);
					homeToSensor := 13;
			END_CASE
					
			//Homing Sensor trigger (torque)
			IF fbMotorHome.Execute AND NOT bHomeSensorTriggered THEN
				bDummyHomingCam := bHomeSensor;
				IF bHomeSensor THEN
					bHomeSensorTriggered := TRUE;
				END_IF
				
			ELSE
				IF stHomingOptions.SearchDirection = MC_Negative_Direction THEN
					fbFreeSensorTimer.IN := TRUE;
					IF fbFreeSensorTimer.Q THEN
						bDummyHomingCam := FALSE;
					END_IF
				ELSE
					bDummyHomingCam := bHomeSensor;
				END_IF
			END_IF
			
			bMotorHomeStatus := fbMotor.Status.Homed;
		END_IF
	ELSE
		fPosition := 0;
		fbMotorMoveAbsolute.Execute := TRUE;
		CASE checkOutputs(stMotorMoveAbsoluteOut) OF 
			1:// Done
				fbMotorMoveAbsolute.Execute := FALSE;
				bHomeSensorTriggered := FALSE;
				fbFreeSensorTimer(IN := FALSE);
				homeToSensor := 1;
			2:// Active
				homeToSensor := 2;
			3:// Busy
			4:// Command Aborted
				fbMotorMoveAbsolute.Execute := FALSE;
			13:// Error
				stError.errorState := MCMOVEABSOLUTE;
				stError.errorLoc := 'homeToSensor_0';
				setError(stMotorMoveAbsoluteOut);
				homeToSensor := 13;
				fbMotorMoveAbsolute.Execute := FALSE;
		END_CASE
	END_IF
END_IF
END_METHOD

METHOD homeToSensorCustom : INT //0:Not done, 1:done, 2:Active, 13: error
VAR_INPUT
END_VAR

(* Need to figure out torque value for homing.
Need to determine which direction of travel to enable*)
////////////////////////////////////////////////////////////
bIdle := FALSE;
IF bIdleDisabled THEN
	IF NOT bMotorHomeStatus THEN
		homeToSensorCustom := 0;
		
		IF bMotorInverted THEN
			direction := 0;
		ELSE 
			direction := 1;
		END_IF
		
		fbhomeToSensorCustom.Execute := TRUE;
		CASE checkOutputs(stHomeToSensorCustomOut) OF 
			1:// Done
				fbHomeToSensorCustom.Execute := FALSE;
				bMotorHomeStatus := fbMotor.Status.Homed;
				homeToSensorCustom := 1; 
			2:// Active
				homeToSensorCustom := 2;
			3:// Busy
				homeToSensorCustom := 3;
			4:// Command Aborted
			13:// Error
				stError.errorState := MCHOME;
				stError.errorLoc := 'homeToSensorCustom';
				setError(stHomeToSensorCustomOut);
				homeToSensorCustom := 13;
		END_CASE
	ELSE
		CASE nHomeState OF 
			0: // Read soft limit switch to set home pos. 
				IF bMotorInverted THEN
					eParameter := AxisMaxSoftPosLimit;
				ELSE 
					eParameter := AxisMinSoftPosLimit;
				END_IF
				
				fbReadRealParam.Enable := TRUE;
				
				IF NOT stReadParamOut.Busy AND stReadParamOut.Done THEN
					fbReadRealParam.Enable := FALSE;
					fPosition := fReadValue;
					nHomeState := nHomeState + 1;
				ELSIF NOT stReadParamOut.Busy AND stReadParamOut.Error THEN
					homeToSensorCustom := 13;
					fbReadRealParam.Enable := FALSE;
					nHomeState := 0;
				END_IF
		
			1: // Execute Move to Home Pos. 
			
			fbMotorMoveAbsolute.Execute := TRUE;
			CASE checkOutputs(stMotorMoveAbsoluteOut) OF 
				1:// Done
					fbMotorMoveAbsolute.Execute := FALSE;
					nHomeState := 0;
					homeToSensorCustom := 1;
				2:// Active
					homeToSensorCustom := 2;
				3:// Busy
					homeToSensorCustom := 3;
				4:// Command Aborted
					fbMotorMoveAbsolute.Execute := FALSE;
					nHomeState := 0;
				13:// Error
					stError.errorState := MCMOVEABSOLUTE;
					stError.errorLoc := 'homeToSensorCustom_0';
					setError(stMotorMoveAbsoluteOut);
					nHomeState := 0;
					homeToSensorCustom := 13;
			END_CASE
		END_CASE
	END_IF
END_IF
END_METHOD

METHOD homeToTorque : INT //0:Not done, 1:done, 2:Active, 13: error
VAR_INPUT
END_VAR

(* Need to figure out torque value for homing.
Need to determine which direction of travel to enable*)
////////////////////////////////////////////////////////////
bIdle := FALSE;
IF bIdleDisabled THEN
	IF NOT bMotorHomeStatus THEN
		homeToTorque := 0;
		
		IF bMotorInverted THEN
			direction := 0;
		ELSE 
			direction := 1;
		END_IF
		
		fbHomeToTorque.Execute := TRUE;
		CASE checkOutputs(stHomeToTorqueOut) OF 
			1:// Done
				fbHomeToTorque.Execute := FALSE;
				bMotorHomeStatus := fbMotor.Status.Homed;
				homeToTorque := 1; 
			2:// Active
				homeToTorque := 2;
			3:// Busy
				homeToTorque := 3;
			4:// Command Aborted
			13:// Error
				stError.errorState := MCHOME;
				stError.errorLoc := 'homeToTorque';
				setError(stHomeToTorqueOut);
				homeToTorque := 13;
		END_CASE
	ELSE
		CASE nHomeState OF 
			0: // Read soft limit switch to set home pos. 
				IF bMotorInverted THEN
					eParameter := AxisMaxSoftPosLimit;
				ELSE 
					eParameter := AxisMinSoftPosLimit;
				END_IF
				
				fbReadRealParam.Enable := TRUE;
				
				IF NOT stReadParamOut.Busy AND stReadParamOut.Done THEN
					fbReadRealParam.Enable := FALSE;
					fPosition := fReadValue;
					nHomeState := nHomeState + 1;
				ELSIF NOT stReadParamOut.Busy AND stReadParamOut.Error THEN
					homeToTorque := 13;
					fbReadRealParam.Enable := FALSE;
					nHomeState := 0;
				END_IF
		
			1: // Execute Move to Home Pos. 
			
			fbMotorMoveAbsolute.Execute := TRUE;
			CASE checkOutputs(stMotorMoveAbsoluteOut) OF 
				1:// Done
					fbMotorMoveAbsolute.Execute := FALSE;
					nHomeState := 0;
					homeToTorque := 1;
				2:// Active
					homeToTorque := 2;
				3:// Busy
					homeToTorque := 3;
				4:// Command Aborted
					fbMotorMoveAbsolute.Execute := FALSE;
					nHomeState := 0;
				13:// Error
					stError.errorState := MCMOVEABSOLUTE;
					stError.errorLoc := 'homeToTorque_0';
					setError(stMotorMoveAbsoluteOut);
					nHomeState := 0;
					homeToTorque := 13;
			END_CASE
		END_CASE
	END_IF
END_IF
END_METHOD

METHOD init : BOOL
VAR_INPUT
	bMotorInvertedIn : BOOL; //True if movement away from home position increases counts negatively
	bMotorDisablesIn : BOOL; //True if motor has a brake attached or does not to be enabled when not moving. 
	
	fMoveAcclIn 		: LREAL;
	fMoveDclIn 			: LREAL;
	fMoveVelocityIn 	: LREAL;
	
	torqueVelocityIn		: LREAL;
	torqueAccelerationIn	: LREAL;
	torqueDecelerationIn	: LREAL;
	
	homeVelocityIn			: LREAL; //Homing velocity when homing when using homeToTorque method.
	homeSetPositionIn		: LREAL; //Counts to set encoder when any homing method is complete. 
	homeTorqueLimitIn		: LREAL; //Torque limit to home to when using homeToTorque method. 
	
	jogTorqueIn				: LREAL; // Torque used to limit jog moves. 
	
	bHasHomeSensorIn		:BOOL; // Does this motor have a homing sensor to home to?  
END_VAR
init := FALSE;
CASE nInitState OF 
	0: //Reset all function blocks 
		IF resetMotorCommands() THEN
			fbMotorPower.Enable := FALSE;
			nInitState := 5;
		END_IF
	5: // Enable Motor
		CASE enable() OF 
			1:// Done
				nInitState := 6;
			2:// Busy	
			13:// Error
				SetError(stMotorPowerOut);
				stError.errorState := MCPOWER;
				nInitState := 10;
		END_CASE
	6: //Set Init Vars
		bMotorInverted := bMotorInvertedIn;
		bMotorDisables := bMotorDisablesIn;
		
		fMoveAccl 		:= fMoveAcclIn;
		fMoveDcl 		:= fMoveDclIn;
		fMoveVelocity 	:= fMoveVelocityIn;
    	
		torqueVelocity		:= torqueVelocityIn;
		torqueAcceleration	:= torqueAccelerationIn;
		torqueDeceleration	:= torqueDecelerationIn;
		
		homeVelocity		:= homeVelocityIn;
		
		homeSetPosition		:= homeSetPositionIn;
		homeTorqueLimit		:= homeTorqueLimitIn;
		
		jogTorque := jogTorqueIn;
		
		bHasHomeSensor := bHasHomeSensorIn;
		
		IF NOT bMotorInverted THEN
			stHomingOptions.SearchDirection := MC_Negative_Direction;
		END_IF
		
		nInitState := 0;
		init := TRUE;
		
	7:// Write homing velocity
	
	
	10:// Error			
		CASE reset() OF 
			1:// Done
				nInitState := 0;
			13:// Error
				nInitState := 0;
		END_CASE
END_CASE
END_METHOD

PROPERTY isBusy : BOOL
GET
isBusy := fbMotor.Status.HasJob;
END_GET
END_PROPERTY

PROPERTY isEnabled : BOOL
GET
isEnabled := NOT fbMotor.Status.Disabled;
END_GET
END_PROPERTY

PROPERTY isMotorInverted : BOOL
GET
isMotorInverted := bMotorInverted;
END_GET
END_PROPERTY

PROPERTY isStopped : BOOL
GET
isStopped := fbMotor.Status.HasBeenStopped;
END_GET
END_PROPERTY

PROPERTY stMotorError : ST_errorRef
GET
motorError.errorId := stError.errorId;
motorError.errorLoc := stError.errorLoc;
motorerror.errorMsg := stError.errorMsg;
motorError.errorState := stError.errorState;
END_GET
END_PROPERTY

PROPERTY motorErrorId : UDINT
GET
motorErrorId := stError.errorId;
END_GET
END_PROPERTY

PROPERTY motorIdle : BOOL
SET
bIdle := motorIdle;
END_SET
END_PROPERTY

METHOD moveTo : INT //0: move not done, 1: Move done, 13: error, 15: move is halway complete
VAR_INPUT
	sState 		: STRING; // *OPTIONAL. Can be used to set the state of the move function (0 is reset, 'NULL' is do nothing);
	fHeightInput : REAL;
END_VAR
//////////////////////////////////////////////////////////////////

IF sState = 'NULL' THEN 
	//Do nothing
ELSE
	nMoveState := STRING_TO_INT(sState);
END_IF
moveTo := 0;
fHeightInput := fHeightInput * 25.4; //Convert inches to mm. 
IF bMotorInverted THEN
	fHeightInput := -fHeightInput;
END_IF

bIdle := FALSE;
IF bIdleDisabled THEN
	CASE nMoveState OF 
		0:// Get Average height of sensor 
			fPosition := fHeightInput;
			fStartPos := fbMotor.NcToPlc.ActPos;
			fHalfwayPos := fStartPos + ((fPosition-fStartPos)*0.75);
			nMoveState := 1;
		
		1:// Execute Move
			fPosition := fHeightInput;
			fbMotorMoveAbsolute.Execute := TRUE;
			CASE checkOutputs(stMotorMoveAbsoluteOut) OF 
				1:// Done
					IF fbMotor.NcToPlc.ActPos < fHeightInput + 1 OR fbMotor.NcToPlc.ActPos > fHeightInput - 1 THEN
						fbMotorMoveAbsolute.Execute := FALSE;
						nMoveState := 0;
						moveTo := 1;
					END_IF
				2,3:// Active,Busy
					moveTo := 2;
					IF ABS(fbMotor.NcToPlc.ActPos) >= ABS(fHalfwayPos) THEN
						moveTo := 15;
					END_IF 
				4:// Command Aborted
					fbMotorMoveAbsolute.Execute := FALSE;
				13:// Error
					stError.errorState := MCMOVEABSOLUTE;
					stError.errorLoc := 'MoveTo';
					setError(stMotorMoveAbsoluteOut);
					nMoveState := 0;
					moveTo := 13;
			END_CASE
			(*IF ABS(fbMotor.NcToPlc.ActPos) >= ABS(fHalfwayPos) THEN
				moveTo := 15;
			END_IF *)
	END_CASE
END_IF
END_METHOD

METHOD moveToJog : INT
VAR_INPUT
	nDirection		: INT; // 0- Negative Moves, 1- Positive Moves
END_VAR
moveToJog := 0;

bIdle := FALSE;
IF bIdleDisabled THEN
	eJogMode := MC_JOGMODE_CONTINOUS;
	fbMotorJog.JogForward := SEL(nDirection = 1,FALSE,TRUE);
	fbMotorJog.JogBackwards := SEL(nDirection = 1,TRUE,FALSE);
	
	CASE checkOutputs(stMotorJogOut) OF 
		1:// Done
		2,3:// Active or Busy	
			moveToJog := 1;
		4:// Command Aborted
		13:// Error
			stError.errorState := MCJOG;
			stError.errorLoc := 'MoveToJog';
			setError(stMotorJogOut);
			moveToJog := 13;
	END_CASE 
END_IF
END_METHOD

METHOD moveToSensor : INT
VAR_INPUT
	nDirection		: INT; // 0- Negative Moves, 1- Positive Moves
END_VAR
moveToSensor := 0;

bIdle := FALSE;
IF bIdleDisabled THEN
	eJogMode := MC_JOGMODE_CONTINOUS;
	fbMotorJog.JogForward := SEL(nDirection = 1,FALSE,TRUE);
	fbMotorJog.JogBackwards := SEL(nDirection = 1,TRUE,FALSE);
	CASE checkOutputs(stMotorJogOut) OF 
		1:// Done
		2,3:// Active or Busy
			IF bClampSensor THEN
				fbMotorJog.JogForward := FALSE;
				fbMotorJog.JogBackwards := FALSE;
				moveToSensor := 1;
			END_IF
		4:// Command Aborted
		13:// Error
			stError.errorState := MCJOG;
			stError.errorLoc := 'MoveToSensor';
			setError(stMotorJogOut);
			moveToSensor := 13;
	END_CASE 
END_IF
END_METHOD

METHOD moveToTorque : INT
VAR_INPUT
	sState 			: STRING; // *OPTIONAL. Can be used to set the state of the move function (0 is reset, 'NULL' is do nothing);
	fTorqueInput 	: REAL; // Percentage of torque to move to.
	nDirection		: INT; //// 0- PositiveDirection, 1- NegativeDirection
END_VAR
IF sState = 'NULL' THEN 
	//Do nothing
ELSE
	nMoveStateTorque := STRING_TO_INT(sState);
END_IF
moveToTorque := 0;
torqueDirection := nDirection;

bIdle := FALSE;
IF bIdleDisabled THEN
	CASE nMoveStateTorque OF 
		0:// Set Torque 
			fTorque := fTorqueInput;
			fbMotorTorque.Execute := FALSE;
			nMoveStateTorque := 1;
			
		1:// Execute Move
			fbMotorTorque.Execute := TRUE;
			CASE checkOutputs(stMotorTorqueOut) OF 
				1:// Done
					fbMotorTorque.Execute := FALSE;
					nMoveStateTorque := 0;
					moveToTorque := 1;
				2:// Active
					moveToTorque := 2;
				3:// Busy
				4:// Command Aborted
					fbMotorTorque.Execute := FALSE;
				13:// Error
					stError.errorState := MCTORQUECONTROL;
					stError.errorLoc := 'MoveToTorque';
					setError(stMotorTorqueOut);
					nMoveStateTorque := 0;
					moveToTorque := 13;
			END_CASE
	END_CASE
END_IF
END_METHOD

METHOD readRealParameter : INT
VAR_INPUT
	parameterIn : MC_AxisParameter; 
END_VAR
readRealParameter := 0;
eParameter := parameterIn;
fbReadRealParam.Enable := TRUE;

CASE checkOutputs(stReadParamOut) OF 	
	1:// Done
		readRealParameter := 1;
	3:// Busy 
		readRealParameter := 2;
	13:// Error
		readRealParameter := 13;	
END_CASE
END_METHOD

METHOD removeStop : INT
VAR_INPUT
END_VAR
removeStop := 0;
IF bMotorDisables THEN
	CASE enable() OF 
		1: // Done
			fbMotorStop.Execute := FALSE;
			IF NOT stMotorStopOut.Busy AND NOT stMotorStopOut.Active THEN 
				brakeOff();
				fbMotorStop.Execute := FALSE;
				removeStop := 1;
			ELSIF stMotorHaltOut.Error THEN
				stError.errorState := MCSTOP;
				stError.errorLoc :=  'teknicMotorHeight_removeStop';
				setError(stMotorStopOut);
				removeStop := 13;
			END_IF
		2: //Busy
		13: //Error
			stError.errorState := MCPOWER;
			stError.errorLoc :=  'teknicMotorHeight_removeStop';
			setError(stMotorPowerOut);
			removeStop := 13;
	END_CASE
ELSE
	fbMotorStop.Execute := FALSE;
IF NOT fbMotor.Status.MotionCommandsLocked THEN
	removeStop := 1;
END_IF

CASE checkOutputs(stMotorPowerOut) OF 
	13:// Error
		removeStop := 13;
END_CASE
END_IF
END_METHOD

METHOD reset : INT //0: reset not done, 1: reset done, 2: Busy, 13: error 
VAR_INPUT
END_VAR
reset := 0;
CASE nResetState OF 
	0: // Remove executes on all motor commands
		resetMotorCommands();
		//bMotorHomeStatus := FALSE;
		nResetState := 3;
	3:// Uncouple Motor
		IF fbMotor.Status.Coupled THEN
			nResetState := 4;
		ELSE
			nResetState := 5;
		END_IF
	4:// Decouple Motor
		CASE decoupleAxis() OF 
			1: // Done
				nResetState := 5;
			13: //Error
				nResetState := 0;
				reset := 13;
		END_CASE
	5://Reset Motor
		fbMotorReset.Execute := TRUE;
		CASE checkOutputs(stMotorResetOut) OF 
			1:// Done
				nResetState := 10;
				fbMotorReset.Execute := FALSE;
			2://Active 
				reset := 2;
			3:// Busy
				reset := 2;
			13:// Error
				setError(stMotorResetOut);
				stError.errorState := MCRESET;
				nResetState := 0;
				reset := 13;
		END_CASE
		
	10: //Motor Off 
		IF stMotorPowerOut.Done OR stMotorPowerOut.Error THEN
			fbMotorPower.Enable := FALSE;
			nResetState := 15;
		ELSE
			nResetState := 15;
		END_IF
		
	15://Power Motor On
		fbMotorPower.Enable := TRUE;
		CASE checkOutputs(stMotorPowerOut) OF
			1: //Done
				nResetState := 0;
				reset := 1;
			13: nResetState := 0;
		END_CASE
	
END_CASE
END_METHOD

METHOD resetMotorCommands : BOOL
VAR_INPUT
END_VAR
resetMotorCommands				:= FALSE;
fbMotorReset.Execute 			:= FALSE;
fbMotorHome.Execute 			:= FALSE;
fbMotorReadMode.Execute  		:= FALSE;
fbMotorWriteMode.Execute 		:= FALSE;
fbMotorHalt.Execute      		:= FALSE;
fbMotorStop.Execute      		:= FALSE;
fbMotorMoveAbsolute.Execute 	:= FALSE;
fbMotorMoveVelocity.Execute 	:= FALSE;
fbMotorMoveRelative.Execute 	:= FALSE;
fbMotorTorque.Execute			:= FALSE;
fbMotorGearIn.Execute			:= FALSE;
fbMotorGearOut.Execute			:= FALSE;
fbMotorJog.JogForward 			:= FALSE;
fbMotorJog.JogBackwards 		:= FALSE;
fbHomeToTorque.Execute			:= FALSE;
fbReadRealParam.Enable 			:= FALSE;
fbWriteRealParam.Execute		:= FALSE;

//Reset FB states
nMoveState 		 := 0;
nMoveStateTorque := 0;
nHomeState		 := 0;
nInitState 		 := 0;
estopState		 := 0;
stopState		 := 0;
resetMotorCommands				:= TRUE;
END_METHOD

METHOD setError : BOOL
VAR_INPUT
	stOutput : REFERENCE TO ST_MCOUTPUTS;
END_VAR
stError.errorId := stOutput.ErrorID;
brakeOn();
END_METHOD

METHOD stop : INT //0: stop not done, 1: stop done; 13: error
VAR_INPUT
END_VAR
(*stop := 0;
fbMotorJog.JogForward 	:= FALSE;
fbMotorJog.JogBackwards := FALSE;
IF stMotorPowerOut.Done THEN
	fbMotorStop.Execute := TRUE;
	fbMotorGearOut.Execute := TRUE;
	CASE checkOutputs(stMotorStopOut) OF 
		1:// Done
			fbMotorGearOut.Execute := FALSE;
			IF bMotorDisables THEN
				brakeOn();
				fbMotorPower.Enable := FALSE;
			END_IF
			stop := 1;
		2:// Active
		3:// Busy
		4:// Command Aborted
		13:// Error
			stError.errorState := MCSTOP;
			stError.errorLoc := 'Height Motor Stop';
			setError(stMotorStopOut);
			stop := 13;
	END_CASE
ELSE
	fbMotorStop.Execute := FALSE;
	stop := 1;
END_IF
*)
stop := 0;
fbMotorJog.JogForward  := FALSE;
fbMotorJog.JogBackwards := FALSE;

CASE stopState OF
    0: // Wait for motor power confirmation
        IF stMotorPowerOut.Done THEN
            fbMotorGearOut.Execute := FALSE;
			fbMotorGearIn.Execute := FALSE;
            stopState := 1;
        ELSE
            stop := 1;
        END_IF

    1: // Wait for GearOut
		fbMotorGearOut.Execute := TRUE;
        IF fbMotorGearOut.Done THEN
            fbMotorGearOut.Execute := FALSE;
            fbMotorStop.Execute := FALSE;
            stopState := 2;
        END_IF

    2: // Wait for Stop
		fbMotorStop.Execute := TRUE;
        CASE checkOutputs(stMotorStopOut) OF 
            1: // Done
                fbMotorStop.Execute := FALSE;
				IF bMotorDisables THEN
            		brakeOn();
                	fbMotorPower.Enable := FALSE;
            	END_IF
				stop := 1;
            	stopState := 0;

            13: // Error
                stError.errorState := MCSTOP;
                stError.errorLoc := 'Height Motor Stop';
                setError(stMotorStopOut);
                stop := 13;
                stopState := 0;
        END_CASE

END_CASE
END_METHOD

METHOD tempCylinderClose : BOOL
VAR_INPUT
END_VAR
tempCylinderClose := FALSE;
bTempCylinder := FALSE;
tempCylinderClose := TRUE;
END_METHOD

METHOD tempCylinderOpen : BOOL
VAR_INPUT
END_VAR
tempCylinderOpen := FALSE;
bTempCylinder := TRUE;
tempCylinderOpen := TRUE;
END_METHOD

METHOD writeRealParameter : INT
VAR_INPUT
	parameterIn : MC_AxisParameter;
	valueIn : LREAL;
END_VAR
writeRealParameter := 0;
eParameter := parameterIn;
fWriteValue := valueIn;
fbWriteRealParam.Execute := TRUE;

CASE checkOutputs(stWriteParameterOut) OF 	
	1:// Done
		writeRealParameter := 1;
	3:// Busy 
		writeRealParameter := 2;
	13:// Error
		writeRealParameter := 13;	
END_CASE
END_METHOD

END_FUNCTION_BLOCK

// ---- POUs/FUNCTIONS/FB_moveToTorque.TcPOU
FUNCTION_BLOCK FB_moveToTorque
VAR_IN_OUT
	Axis : AXIS_REF;					
END_VAR
VAR_INPUT
	Execute 			: BOOL;
	Direction 			: INT; // 0- PositiveDirection, 1- NegativeDirection
	Velocity 			: LREAL;
	Acceleration 		: LREAL;
	Deceleration 		: LREAL;
	DetectionTorqueTime : TIME;
	TorqueLimit 		: LREAL;
END_VAR
VAR_OUTPUT
	Done 			: BOOL;
	Busy 			: BOOL;
	Active 			: BOOL;
	CommandAborted 	: BOOL;
	Error 			: BOOL;
	ErrorID 		: UDINT;
END_VAR
VAR
	nState 			: INT;
	fbExecute 		: R_TRIG;
	fbDetectTime 	: TON;
	
	readParameter 		: MC_ReadParameter;
	readParameterOut 	: ST_mcOutputs;
	
	writeParameter		: MC_WriteParameter;
	writeParameterOut 	: ST_mcOutputs;
	readValue 			: LREAL;
	
	parameter 	: MC_AxisParameter;	
	writeValue 	: LREAL;
	
	moveToTorque	: MC_TorqueControl;
	torqueOptions 	: ST_TorqueControlOptions;
	moveToTorqueOut : ST_mcOutputs;
	
	moveAbsolute	: MC_MoveAbsolute;
	moveAbsoluteOut : ST_mcOutputs;
	calcBackOffPos 	: LREAL;
	
	home	: MC_Home;
	homeOut : ST_mcOutputs;
	
	stop		: MC_Stop;
	stopOut 	: ST_mcOutputs;
	fPosition	: LREAL;

	jog		: MC_Jog;
	jogOut 	: ST_mcOutputs;
	
	moveRelative	: MC_MoveRelative;
	moveRelativeOut	: ST_mcOutputs;
END_VAR

fbExecute(CLK := Execute);
fbDetectTime.PT := DetectionTorqueTime;
fbDetectTime();
actMove();


CASE nState OF 
	0: //init
		IF NOT Execute THEN
		(* reset at falling edge of Execute *)
			Busy 					:= FALSE;
			Done					:= FALSE;
			CommandAborted 			:= FALSE;
			Error 					:= FALSE;
			ErrorID 				:= 0;
			fbDetectTime.IN 		:= FALSE;
			readParameter.Enable 	:= FALSE;
			writeParameter.Execute 	:= FALSE;
			stop.Execute 			:= FALSE;
			home.Execute 			:= FALSE;
			moveAbsolute.Execute 	:= FALSE;
			jog.JogForward 			:= FALSE;
			jog.JogBackwards 		:= FALSE;
		END_IF
	
		IF fbExecute.Q THEN
			Busy := TRUE;
			nState := nState + 1;
		END_IF
		
	1: //Execute MoveTowards Torque
		CASE Direction OF
			0: //mcPositiveDirection
				jog.JogForward := TRUE;
				jog.JogBackwards := FALSE;
			1: //mcNegativeDirection
				jog.JogForward := FALSE;
				jog.JogBackwards := TRUE;
		END_CASE
			
